(* POU STP, ST *)
PROGRAM STP
VAR
	LSL100A_MixerFloatSensor AT %I* : BOOL;
	LSH100A_MixerFloatSensor AT %I* : BOOL;
	LSH101A_EQFloatSensor AT %I* : BOOL;
	LSHH101A_EQFloatSensor AT %I* : BOOL;
	LSL101A_EQFloatSensor AT %I* : BOOL;
	LSH105A1_StreamLineFlow AT %I* : BOOL;
	LSHH105A2_StreamLineOverflow AT %I* : BOOL;
	LSL103A_SBRFloatSensor AT %I* : BOOL;
	LSHH103A_SBRFloatSensor AT %I* : BOOL;
	LSH103A_SBRFloatSensor AT %I* : BOOL;
	TMT01_FanStatus AT %I* : BOOL;
	DP01_DoorPanelStatus AT %I* : BOOL;
	LSD101A_EQFloatSensorDry AT %I* : BOOL;
	LSD103A_SBRFloatSensorDry AT %I* : BOOL;
	XV101A1_SolenoidValveSpray_OpenStat AT %I* : BOOL;
	XV101A2_SolenoidValveSpray_OpenStat AT %I* : BOOL;
	XV102A1_ContinuosValveWater_OpenStat AT %I* : BOOL;
	XV100A1_GritRemovalValve_OpenStat AT %I* : BOOL;
	XV100A2_GritRemovalValve_OpenStat AT %I* : BOOL;
	PS101A1_Penstock_OpenStat AT %I* : BOOL;
	PS101A2_Penstock_OpenStat AT %I* : BOOL;
	PS101A1_Penstock_CloseStat AT %I* : BOOL;
	PS101A2_Penstock_CloseStat AT %I* : BOOL;
	XV101A1_SolenoidValveSpray_CloseStat AT %I* : BOOL;
	XV101A2_SolenoidValveSpray_CloseStat AT %I* : BOOL;
	XV102A1_ContinuosValveWater_CloseStat AT %I* : BOOL;
	XV100A1_GritRemovalValve_CloseStat AT %I* : BOOL;
	XV100A2_GritRemovalValve_CloseStat AT %I* : BOOL;
	M101A1_EQMixer_OverloadStat AT %I* : BOOL;
	M101A1_EQMixer_IncompleteStat AT %I* : BOOL;
	M101A2_EQMixer_OverloadStat AT %I* : BOOL;
	M101A2_EQMixer_IncompleteStat AT %I* : BOOL;
	P101A1_EQPump_OverloadStat AT %I* : BOOL;
	P101A1_EQPump_IncompleteStat AT %I* : BOOL;
	P101A2_EQPump_OverloadStat AT %I* : BOOL;
	P101A2_EQPump_IncompleteStat AT %I* : BOOL;
	PS101A1_Penstock_TripStat AT %I* : BOOL;
	PS101A2_Penstock_TripStat AT %I* : BOOL;
	F101A1_FineScr_OverloadStat AT %I* : BOOL;
	F101A2_FineScr_OverloadStat AT %I* : BOOL;
	C102A_ScreeningConveyer_OverloadStat AT %I* : BOOL;
	C101A_ScreeningCompactor_OverloadStat AT %I* : BOOL;
	C103A_GritClassifier_OverloadStat AT %I* : BOOL;
	P102A1_SBRTransferPump_OverloadStat AT %I* : BOOL;
	P102A1_SBRTransferPump_IncompleteStat AT %I* : BOOL;
	P102A2_SBRTransferPump_OverloadStat AT %I* : BOOL;
	P102A2_SBRTransferPump_IncompleteStat AT %I* : BOOL;
	M101A1_EQMixer_LocalRemoteStat AT %I* : BOOL;
	M101A2_EQMixer_LocalRemoteStat AT %I* : BOOL;
	P101A1_EQPump_LocalRemoteStat AT %I* : BOOL;
	P101A2_EQPump_LocalRemoteStat AT %I* : BOOL;
	F101A1_FineScr_LocalRemoteStat AT %I* : BOOL;
	F101A2_FineScr_LocalRemoteStat AT %I* : BOOL;
	C102A_ScreenConveyer_LocalRemoteStat AT %I* : BOOL;
	C101A_ScreenCompactor_LocalRemoteStat AT %I* : BOOL;
	C103A_GritClasifier_LocalRemoteStat AT %I* : BOOL;
	P102A1_SBRTransferPump_LocalRemoteStat AT %I* : BOOL;
	P102A2_SBRTransferPump_LocalRemoteStat AT %I* : BOOL;
	PS101A1_Penstock_LocalRemoteStat AT %I* : BOOL;
	PS101A2_Penstock_LocalRemoteStat AT %I* : BOOL;
	M101A1_EQMixer_RunStat AT %I* : BOOL;
	M101A2_EQMixer_RunStat AT %I* : BOOL;
	P101A1_EQPump_RunStat AT %I* : BOOL;
	P101A2_EQPump_RunStat AT %I* : BOOL;
	F101A1_FineScr_RunStat AT %I* : BOOL;
	F101A2_FineScr_RunStat AT %I* : BOOL;
	C102A_ScreenConveyer_RunStat AT %I* : BOOL;
	C101A_ScreenCompactor_RunStat AT %I* : BOOL;
	C103A_GritClasifier_RunStat AT %I* : BOOL;
	P102A1_SBRTransferPump_RunStat AT %I* : BOOL;
	P102A2_SBRTransferPump_RunStat AT %I* : BOOL;
	M101A1_EQMixer_EStopStat AT %I* : BOOL;
	M101A2_EQMixer_EStopStat AT %I* : BOOL;
	P101A1_EQPump_EStopStat AT %I* : BOOL;
	P101A2_EQPump_EStopStat AT %I* : BOOL;
	F101A1_FineScr_EStopStat AT %I* : BOOL;
	F101A2_FineScr_EStopStat AT %I* : BOOL;
	C102A_ScreenConveyer_EStopStat AT %I* : BOOL;
	C101A_ScreenCompactor_EStopStat AT %I* : BOOL;
	C103A_GritClasifier_EStopStat AT %I* : BOOL;
	P102A1_SBRTransferPump_EStopStat AT %I* : BOOL;
	P102A2_SBRTransferPump_EStopStat AT %I* : BOOL;
	B101A1_AirBlower_OverloadStat AT %I* : BOOL;
	B101A1_AirBlower_IncompleteStat AT %I* : BOOL;
	B101A2_AirBlower_OverloadStat AT %I* : BOOL;
	B101A2_AirBlower_IncompleteStat AT %I* : BOOL;
	B101A1_AirBlower_LocalRemoteStat AT %I* : BOOL;
	B101A2_AirBlower_LocalRemoteStat AT %I* : BOOL;
	B101A1_AirBlower_OnOffStat AT %I* : BOOL;
	B101A2_AirBlower_OnOffStat AT %I* : BOOL;
	B101A1_AirBlower_EStopStat AT %I* : BOOL;
	B101A2_AirBlower_EStopStat AT %I* : BOOL;
	XV101A1_SolenoidValveSpray_OpenCmd AT %Q* : BOOL;
	XV101A2_SolenoidValveSpray_OpenCmd AT %Q* : BOOL;
	XV102A1_ContinuosValveWater_OpenCmd AT %Q* : BOOL;
	F101A1_FineScr_RunCmd AT %Q* : BOOL;
	F101A2_FineScr_RunCmd AT %Q* : BOOL;
	C102A_ScreenConveyer_RunCmd AT %Q* : BOOL;
	C101A_ScreenCompactor_RunCmd AT %Q* : BOOL;
	C103A_GritClasifier_RunCmd AT %Q* : BOOL;
	PS101A1_Penstock_OpenCmd AT %Q* : BOOL;
	PS101A1_Penstock_CloseCmd AT %Q* : BOOL;
	PS101A2_Penstock_OpenCmd AT %Q* : BOOL;
	PS101A2_Penstock_CloseCmd AT %Q* : BOOL;
	XV100A1_GritRemovalValve_OpenCmd AT %Q* : BOOL;
	XV100A2_GritRemovalValve_OpenCmd AT %Q* : BOOL;
	P101A1_EQPump_RunCmd AT %Q* : BOOL;
	P101A2_EQPump_RunCmd AT %Q* : BOOL;
	M101A1_EQMixer_RunCmd AT %Q* : BOOL;
	M101A2_EQMixer_RunCmd AT %Q* : BOOL;
	B101A1_AirBlower_RunCmd AT %Q* : BOOL;
	B101A2_AirBlower_RunCmd AT %Q* : BOOL;
	P102A1_SBRTransferPump_RunCmd AT %Q* : BOOL;
	P102A2_SBRTransferPump_RunCmd AT %Q* : BOOL;
	AUX101A_EQFloatSensor_AlarmS1 AT %Q* : BOOL;
	AUX104A_SBRFloatSensor_AlarmS1 AT %Q* : BOOL;
	AUX105A_StreamSensorOverflow_AlarmS1 AT %Q* : BOOL;
	AUX101_CommonAlarm AT %Q* : BOOL;
	AUX102_PLCRunStat AT %Q* : BOOL;
	LSL100B_MixerFloatSensor AT %I* : BOOL;
	LSH100B_MixerFloatSensor AT %I* : BOOL;
	LSH101B_EQFloatSensor AT %I* : BOOL;
	LSHH101B_EQFloatSensor AT %I* : BOOL;
	LSL101B_EQFloatSensor AT %I* : BOOL;
	LSH105B1_StreamLineFlow AT %I* : BOOL;
	LSHH105B2_StreamLineOverflow AT %I* : BOOL;
	LSH103B_SBRFloatSensor AT %I* : BOOL;
	LSHH103B_SBRFloatSensor AT %I* : BOOL;
	LSL103B_SBRFloatSensor AT %I* : BOOL;
	LSD101B_EQFloatSensorDry AT %I* : BOOL;
	LSD103B_SBRFloatSensorDry AT %I* : BOOL;
	XV101B1_SolenoidValveSpray_OpenStat AT %I* : BOOL;
	XV101B2_SolenoidValveSpray_OpenStat AT %I* : BOOL;
	XV102B1_ContinuosValveWater_OpenStat AT %I* : BOOL;
	XV100B1_GritRemovalValve_OpenStat AT %I* : BOOL;
	XV100B2_GritRemovalValve_OpenStat AT %I* : BOOL;
	PS101B1_Penstock_OpenStat AT %I* : BOOL;
	PS101B2_Penstock_OpenStat AT %I* : BOOL;
	PS101B1_Penstock_CloseStat AT %I* : BOOL;
	PS101B2_Penstock_CloseStat AT %I* : BOOL;
	XV101B1_SolenoidValveSpray_CloseStat AT %I* : BOOL;
	XV101B2_SolenoidValveSpray_CloseStat AT %I* : BOOL;
	XV102B1_ContinuosValveWater_CloseStat AT %I* : BOOL;
	XV100B1_GritRemovalValve_CloseStat AT %I* : BOOL;
	XV100B2_GritRemovalValve_CloseStat AT %I* : BOOL;
	M101B1_EQMixer_OverloadStat AT %I* : BOOL;
	M101B1_EQMixer_IncompleteStat AT %I* : BOOL;
	M101B2_EQMixer_OverloadStat AT %I* : BOOL;
	M101B2_EQMixer_IncompleteStat AT %I* : BOOL;
	P101B1_EQPump_OverloadStat AT %I* : BOOL;
	P101B1_EQPump_IncompleteStat AT %I* : BOOL;
	P101B2_EQPump_OverloadStat AT %I* : BOOL;
	P101B2_EQPump_IncompleteStat AT %I* : BOOL;
	PS101B1_Penstock_TripStat AT %I* : BOOL;
	PSB101B2_Penstock_TripStat AT %I* : BOOL;
	F101B1_FineScr_OverloadStat AT %I* : BOOL;
	F101B2_FineScr_OverloadStat AT %I* : BOOL;
	C102B_ScreeningConveyer_OverloadStat AT %I* : BOOL;
	C101B_ScreeningCompactor_OverloadStat AT %I* : BOOL;
	C103B_GritClassifier_OverloadStat AT %I* : BOOL;
	P102B1_SBRTransferPump_OverloadStat AT %I* : BOOL;
	P102B1_SBRTransferPump_IncompleteStat AT %I* : BOOL;
	P102B2_SBRTransferPump_OverloadStat AT %I* : BOOL;
	P102B2_SBRTransferPump_IncompleteStat AT %I* : BOOL;
	M101B1_EQMixer_LocalRemoteStat AT %I* : BOOL;
	M101B2_EQMixer_LocalRemoteStat AT %I* : BOOL;
	P101B1_EQPump_LocalRemoteStat AT %I* : BOOL;
	P101B2_EQPump_LocalRemoteStat AT %I* : BOOL;
	F101B1_FineScr_LocalRemoteStat AT %I* : BOOL;
	F101B2_FineScr_LocalRemoteStat AT %I* : BOOL;
	C102B_ScreenConveyer_LocalRemoteStat AT %I* : BOOL;
	C101B_ScreenCompactor_LocalRemoteStat AT %I* : BOOL;
	C103BB_GritClasifiier_LocalRemoteStat AT %I* : BOOL;
	P102B1_SBRTransferPump_LocalRemoteStat AT %I* : BOOL;
	P102B2_SBRTransferPump_LocalRemoteStat AT %I* : BOOL;
	PS101B1_Penstock_LocalRemoteStat AT %I* : BOOL;
	PS101B2_Penstock_LocalRemoteStat AT %I* : BOOL;
	M101B1_EQMixer_RunStat AT %I* : BOOL;
	M101B2_EQMixer_RunStat AT %I* : BOOL;
	P101B1_EQPump_RunStat AT %I* : BOOL;
	P101B2_EQPump_RunStat AT %I* : BOOL;
	F101B1_FineScr_RunStat AT %I* : BOOL;
	F101B2_FineScr_RunStat AT %I* : BOOL;
	C102B_ScreenConveyer_RunStat AT %I* : BOOL;
	C101B_ScreenCompactor_RunStat AT %I* : BOOL;
	C103B_GritClasifier_RunStat AT %I* : BOOL;
	P102B1_SBRTransferPump_RunStat AT %I* : BOOL;
	P102B2_SBRTransferPump_RunStat AT %I* : BOOL;
	M101B1_EQMixer_EStopStat AT %I* : BOOL;
	M101B2_EQMixer_EStopStat AT %I* : BOOL;
	P101B1_EQPump_EStopStat AT %I* : BOOL;
	P101B2_EQPump_EStopStat AT %I* : BOOL;
	F101B1_FineScr_EStopStat AT %I* : BOOL;
	F101B2_FineScr_EStopStat AT %I* : BOOL;
	C102B_ScreenConveyer_EStopStat AT %I* : BOOL;
	C101B_ScreenCompactor_EStopStat AT %I* : BOOL;
	C103B_GritClasifier_EStopStat AT %I* : BOOL;
	P102B1_SBRTransferPump_EStopStat AT %I* : BOOL;
	P102B2_SBRTransferPump_EStopStat AT %I* : BOOL;
	VE801A_SuctionFan_OnOffStat AT %I* : BOOL;
	P802A_CirculationPump_OnOffStat AT %I* : BOOL;
	P803A_CirculationPump_OnOffStat AT %I* : BOOL;
	P804A_CirculationPump_OnOffStat AT %I* : BOOL;
	P805A1_H2S04Pump_OnOffStat AT %I* : BOOL;
	P805A2_H2S04Pump_OnOffStat AT %I* : BOOL;
	P806A1_NAOHPump_OnOffStat AT %I* : BOOL;
	P806A2_NAOHPump_OnOffStat AT %I* : BOOL;
	P807A1_NAOCLPump_OnOffStat AT %I* : BOOL;
	P807A2_NAOCLPump_OnOffStat AT %I* : BOOL;
	VE801A_SuctionFan_OverloadStat AT %I* : BOOL;
	P802A_CirculationPump_OverloadStat AT %I* : BOOL;
	P803A_CirculationPump_OverloadStat AT %I* : BOOL;
	P804A_CirculationPump_OverloadStat AT %I* : BOOL;
	P805A1_H2S04Pump_OverloadStat AT %I* : BOOL;
	P805A2_H2S04Pump_OverloadStat AT %I* : BOOL;
	P806A1_NAOHPump_OverloadStat AT %I* : BOOL;
	P806A2_NAOHPump_OverloadStat AT %I* : BOOL;
	P807A1_NAOCLPump_OverloadStat AT %I* : BOOL;
	P807A2_NAOCLPump_OverloadStat AT %I* : BOOL;
	VE801A_SuctionFan_EStopStat AT %I* : BOOL;
	P802A_CirculationPump_EStopStat AT %I* : BOOL;
	P803A_CirculationPump_EStopStat AT %I* : BOOL;
	P804A_CirculationPump_EStopStat AT %I* : BOOL;
	P805A1_H2S04Pump_EStopStat AT %I* : BOOL;
	P805A2_H2S04Pump_EStopStat AT %I* : BOOL;
	P806A1_NAOHPump_EStopStat AT %I* : BOOL;
	P806A2_NAOHPump_EStopStat AT %I* : BOOL;
	P807A1_NAOCLPump_EStopStat AT %I* : BOOL;
	P807A2_NAOCLPump_EStopStat AT %I* : BOOL;
	XV101B1_SolenoidValveSpray_OpenCmd AT %Q* : BOOL;
	XV101B2_SolenoidValveSpray_OpenCmd AT %Q* : BOOL;
	XV102B1_ContinuosValveWater_OpenCmd AT %Q* : BOOL;
	F101B1_FineScr_RunCmd AT %Q* : BOOL;
	F101B2_FineScr_RunCmd AT %Q* : BOOL;
	C102B_ScreenConveyer_RunCmd AT %Q* : BOOL;
	C101B_ScreenCompactor_RunCmd AT %Q* : BOOL;
	C103B_GritClasifier_RunCmd AT %Q* : BOOL;
	PS101B1_Penstock_OpenCmd AT %Q* : BOOL;
	PS101B1_Penstock_CloseCmd AT %Q* : BOOL;
	PS101B2_Penstock_OpenCmd AT %Q* : BOOL;
	PS101B2_Penstock_CloseCmd AT %Q* : BOOL;
	XV100B1_GritRemovalValve_OpenCmd AT %Q* : BOOL;
	XV100B2_GritRemovalValve_OpenCmd AT %Q* : BOOL;
	P101B1_EQPump_RunCmd AT %Q* : BOOL;
	P101B2_EQPump_RunCmd AT %Q* : BOOL;
	M101B1_EQMixer_RunCmd AT %Q* : BOOL;
	M101B2_EQMixer_RunCmd AT %Q* : BOOL;
	P102B1_SBRTransferPump_RunCmd AT %Q* : BOOL;
	P102B2_SBRTransferPump_RunCmd AT %Q* : BOOL;
	AUX101B_EQFloatSensor_AlarmS2 AT %Q* : BOOL;
	AUX104B_SBRFloatSensor_AlarmS2 AT %Q* : BOOL;
	AUX105B_StreamSensorOverflow_AlarmS2 AT %Q* : BOOL;
	TMT02_FanStatus AT %I* : BOOL;
	DP02_DoorPanelStatus AT %I* : BOOL;
	XV261A_DecanterR1_OverloadStat AT %I* : BOOL;
	XV262A_DecanterR2_OverloadStat AT %I* : BOOL;
	XV263A_DecanterR3_OverloadStat AT %I* : BOOL;
	XV264A_DecanterR4_OverloadStat AT %I* : BOOL;
	M200A1A_MixerR1_RunStat AT %I* : BOOL;
	M200A1B_MixerR1_RunStat AT %I* : BOOL;
	M200A1C_MixerR1_RunStat AT %I* : BOOL;
	M200A2A_MixerR2_RunStat AT %I* : BOOL;
	M200A2B_MixerR2_RunStat AT %I* : BOOL;
	M200A2C_MixerR2_RunStat AT %I* : BOOL;
	M200A3A_MixerR3_RunStat AT %I* : BOOL;
	M200A3B_MixerR3_RunStat AT %I* : BOOL;
	M200A3C_MixerR3_RunStat AT %I* : BOOL;
	M200A4A_MixerR4_RunStat AT %I* : BOOL;
	M200A4B_MixerR4_RunStat AT %I* : BOOL;
	M200A4C_MixerR4_RunStat AT %I* : BOOL;
	B201A1_AirBlowerS1_RunStat AT %I* : BOOL;
	B201A2_AirBlowerS1_RunStat AT %I* : BOOL;
	B201A3_AirBlowerS1_RunStat AT %I* : BOOL;
	M200A1A_MixerR1_LocalRemoteStat AT %I* : BOOL;
	M200A1B_MixerR1_LocalRemoteStat AT %I* : BOOL;
	M200A1C_MixerR1_LocalRemoteStat AT %I* : BOOL;
	M200A2A_MixerR2_LocalRemoteStat AT %I* : BOOL;
	M200A2B_MixerR2_LocalRemoteStat AT %I* : BOOL;
	M200A2C_MixerR2_LocalRemoteStat AT %I* : BOOL;
	M200A3A_MixerR3_LocalRemoteStat AT %I* : BOOL;
	M200A3B_MixerR3_LocalRemoteStat AT %I* : BOOL;
	M200A3C_MixerR3_LocalRemoteStat AT %I* : BOOL;
	M200A4A_MixerR4_LocalRemoteStat AT %I* : BOOL;
	M200A4B_MixerR4_LocalRemoteStat AT %I* : BOOL;
	M200A4C_MixerR4_LocalRemoteStat AT %I* : BOOL;
	B201A1_AirBlowerS1_LocalRemoteStat AT %I* : BOOL;
	B201A2_AirBlowerS1_LocalRemoteStat AT %I* : BOOL;
	B201A3_AirBlowerS1_LocalRemoteStat AT %I* : BOOL;
	XV261A_DecanterR1_LocalRemoteStat AT %I* : BOOL;
	XV262A_DecanterR2_LocalRemoteStat AT %I* : BOOL;
	XV263A_DecanterR3_LocalRemoteStat AT %I* : BOOL;
	XV264A_DecanterR4_LocalRemoteStat AT %I* : BOOL;
	P201A1_DesludgePumpS1_LocalRemoteStat AT %I* : BOOL;
	P201A2_DesludgePumpS1_LocalRemoteStat AT %I* : BOOL;
	P201A1_DesludgePumpS1_RunStat AT %I* : BOOL;
	P201A2_DesludgePumpS1_RunStat AT %I* : BOOL;
	M200A1A_MixerR1_OverloadStat AT %I* : BOOL;
	M200A1A_MixerR1_IncompleteStat AT %I* : BOOL;
	M200A1B_MixerR1_OverloadStat AT %I* : BOOL;
	M200A1B_MixerR1_IncompleteStat AT %I* : BOOL;
	M200A1C_MixerR1_OverloadStat AT %I* : BOOL;
	M200A1C_MixerR1_IncompleteStat AT %I* : BOOL;
	M200A2A_MixerR2_OverloadStat AT %I* : BOOL;
	M200A2A_MixerR2_IncompleteStat AT %I* : BOOL;
	M200A2B_MixerR2_OverloadStat AT %I* : BOOL;
	M200A2B_MixerR2_IncompleteStat AT %I* : BOOL;
	M200A2C_MixerR2_OverloadStat AT %I* : BOOL;
	M200A2C_MixerR2_IncompleteStat AT %I* : BOOL;
	M200A3A_MixerR3_OverloadStat AT %I* : BOOL;
	M200A3A_MixerR3_IncompleteStat AT %I* : BOOL;
	M200A3B_MixerR3_OverloadStat AT %I* : BOOL;
	M200A3B_MixerR3_IncompleteStat AT %I* : BOOL;
	M200A3C_MixerR3_OverloadStat AT %I* : BOOL;
	M200A3C_MixerR3_IncompleteStat AT %I* : BOOL;
	M200A4A_MixerR4_OverloadStat AT %I* : BOOL;
	M200A4A_MixerR4_IncompleteStat AT %I* : BOOL;
	M200A4B_MixerR4_OverloadStat AT %I* : BOOL;
	M200A4B_MixerR4_IncompleteStat AT %I* : BOOL;
	M200A4C_MixerR4_OverloadStat AT %I* : BOOL;
	M200A4C_MixerR4_IncompleteStat AT %I* : BOOL;
	B201A1_AirBlowerS1_OverloadStat AT %I* : BOOL;
	B201A1_AirBlowerS1_IncompleteStat AT %I* : BOOL;
	B201A2_AirBlowerS1_OverloadStat AT %I* : BOOL;
	B201A2_AirBlowerS1_IncompleteStat AT %I* : BOOL;
	B201A3_AirBlowerS1_OverloadStat AT %I* : BOOL;
	B201A3_AirBlowerS1_IncompleteStat AT %I* : BOOL;
	P201A1_DesludgePumpS1_OverloadStatus AT %I* : BOOL;
	P201A2_DesludgePumpS1_OverloadStatus AT %I* : BOOL;
	M200A1A_MixerR1_EStopStat AT %I* : BOOL;
	M200A1B_MixerR1_EStopStat AT %I* : BOOL;
	M200A1C_MixerR1_EStopStat AT %I* : BOOL;
	M200A2A_MixerR2_EStopStat AT %I* : BOOL;
	M200A2B_MixerR2_EStopStat AT %I* : BOOL;
	M200A2C_MixerR2_EStopStat AT %I* : BOOL;
	M200A3A_MixerR3_EStopStat AT %I* : BOOL;
	M200A3B_MixerR3_EStopStat AT %I* : BOOL;
	M200A3C_MixerR3_EStopStat AT %I* : BOOL;
	M200A4A_MixerR3_EStopStat AT %I* : BOOL;
	M200A4B_MixerR3_EStopStat AT %I* : BOOL;
	M200A4C_MixerR3_EStopStat AT %I* : BOOL;
	B201A1_AirBlowerS1_EStopStat AT %I* : BOOL;
	B201A2_AirBlowerS1_EStopStat AT %I* : BOOL;
	B201A3_AirBlowerS1_EStopStat AT %I* : BOOL;
	XV261A_DecanterR1_EStopStat AT %I* : BOOL;
	XV262A_DecanterR2_EStopStat AT %I* : BOOL;
	XV263A_DecanterR3_EStopStat AT %I* : BOOL;
	XV264A_DecanterR4_EStopStat AT %I* : BOOL;
	P201A1_DesludgePumpS1_EStopStat AT %I* : BOOL;
	P201A2_DesludgePumpS1_EStopStat AT %I* : BOOL;
	XV261A_DecanterR1_FwdStat AT %I* : BOOL;
	XV262A_DecanterR2_FwdStat AT %I* : BOOL;
	XV263A_DecanterR3_FwdStat AT %I* : BOOL;
	XV264A_DecanterR4_FwdStat AT %I* : BOOL;
	XV261A_DecanterR1_RvsStat AT %I* : BOOL;
	XV262A_DecanterR2_RvsStat AT %I* : BOOL;
	XV263A_DecanterR3_RvsStat AT %I* : BOOL;
	XV264A_DecanterR4_RvsStat AT %I* : BOOL;
	FT100A_FlowTotalizerS1 AT %IW0 : REAL;
	FT100A_FlowTotalizerS1_ScaledValue:INT;
	M200A1A_MixerR1_RunCmd AT %Q* : BOOL;
	M200A1B_MixerR1_RunCmd AT %Q* : BOOL;
	M200A1C_MixerR1_RunCmd AT %Q* : BOOL;
	M200A2A_MixerR2_RunCmd AT %Q* : BOOL;
	M200A2B_MixerR2_RunCmd AT %Q* : BOOL;
	M200A2C_MixerR2_RunCmd AT %Q* : BOOL;
	M200A3A_MixerR3_RunCmd AT %Q* : BOOL;
	M200A3B_MixerR3_RunCmd AT %Q* : BOOL;
	M200A3C_MixerR3_RunCmd AT %Q* : BOOL;
	M200A4A_MixerR4_RunCmd AT %Q* : BOOL;
	M200A4B_MixerR4_RunCmd AT %Q* : BOOL;
	M200A4C_MixerR4_RunCmd AT %Q* : BOOL;
	XV261A_DecanterR1_FwdCmd AT %Q* : BOOL;
	XV262A_DecanterR2_FwdCmd AT %Q* : BOOL;
	XV263A_DecanterR3_FwdCmd AT %Q* : BOOL;
	XV264A_DecanterR4_FwdCmd AT %Q* : BOOL;
	XV261A_DecanterR1_RvsCmd AT %Q* : BOOL;
	XV262A_DecanterR2_RvsCmd AT %Q* : BOOL;
	XV263A_DecanterR3_RvsCmd AT %Q* : BOOL;
	XV264A_DecanterR4_RvsCmd AT %Q* : BOOL;
	B201A1_AirBlowerS1_RunCmd AT %Q* : BOOL;
	B201A2_AirBlowerS1_RunCmd AT %Q* : BOOL;
	B201A3_AirBlowerS1_RunCmd AT %Q* : BOOL;
	P201A1_DesludgePump_RunCmd AT %Q* : BOOL;
	P201A2_DesludgePump_RunCmd AT %Q* : BOOL;
	AUXA1_ReactorS1R1_OpsStat AT %Q* : BOOL;
	AUXA2_ReactorS1R2_OpsStat AT %Q* : BOOL;
	AUXA3_ReactorS1R3_OpsStat AT %Q* : BOOL;
	AUXA4_ReactorS1R4_OpsStat AT %Q* : BOOL;
	AUXB1_ReactorS2R1_OpsStat AT %Q* : BOOL;
	AUXB2_ReactorS2R2_OpsStat AT %Q* : BOOL;
	AUXB3_ReactorS2R3_OpsStat AT %Q* : BOOL;
	AUXB4_ReactorS2R4_OpsStat AT %Q* : BOOL;
	AUXA5_BlowerS1R1 AT %Q* : BOOL;
	AUXA6_BlowerS1R2 AT %Q* : BOOL;
	AUXA7_BlowerS1R3 AT %Q* : BOOL;
	AUXB5_BlowerS2R1 AT %Q* : BOOL;
	AUXB6_BlowerS2R2 AT %Q* : BOOL;
	AUXB7_BlowerS2R3 AT %Q* : BOOL;
	AUX201_CommonAlarm AT %Q* : BOOL;
	AUX202_PLCRunStat AT %Q* : BOOL;
	TMT03_FanStatus AT %I* : BOOL;
	DP03_DoorPanelStatus AT %I* : BOOL;
	XV261B_DecanterR1_OverloadStat AT %I* : BOOL;
	XV262B_DecanterR2_OverloadStat AT %I* : BOOL;
	XV263B_DecanterR3_OverloadStat AT %I* : BOOL;
	XV264B_DecanterR4_OverloadStat AT %I* : BOOL;
	M200B1A_MixerR1_RunStat AT %I* : BOOL;
	M200B1B_MixerR1_RunStat AT %I* : BOOL;
	M200B1C_MixerR1_RunStat AT %I* : BOOL;
	M200B2A_MixerR2_RunStat AT %I* : BOOL;
	M200B2B_MixerR2_RunStat AT %I* : BOOL;
	M200B2C_MixerR2_RunStat AT %I* : BOOL;
	M200B3A_MixerR3_RunStat AT %I* : BOOL;
	M200B3B_MixerR3_RunStat AT %I* : BOOL;
	M200B3C_MixerR3_RunStat AT %I* : BOOL;
	M200B4A_MixerR4_RunStat AT %I* : BOOL;
	M200B4B_MixerR4_RunStat AT %I* : BOOL;
	M200B4C_MixerR4_RunStat AT %I* : BOOL;
	B201B1_AirBlowerS2_RunStat AT %I* : BOOL;
	B201B2_AirBlowerS2_RunStat AT %I* : BOOL;
	B201B3_AirBlowerS2_RunStat AT %I* : BOOL;
	M200B1A_MixerR1_LocalRemoteStat AT %I* : BOOL;
	M200B1B_MixerR1_LocalRemoteStat AT %I* : BOOL;
	M200B1C_MixerR1_LocalRemoteStat AT %I* : BOOL;
	M200B2A_MixerR2_LocalRemoteStat AT %I* : BOOL;
	M200B2B_MixerR2_LocalRemoteStat AT %I* : BOOL;
	M200B2C_MixerR2_LocalRemoteStat AT %I* : BOOL;
	M200B3A_MixerR3_LocalRemoteStat AT %I* : BOOL;
	M200B3B_MixerR3_LocalRemoteStat AT %I* : BOOL;
	M200B3C_MixerR3_LocalRemoteStat AT %I* : BOOL;
	M200B4A_MixerR4_LocalRemoteStat AT %I* : BOOL;
	M200B4B_MixerR4_LocalRemoteStat AT %I* : BOOL;
	M200B4C_MixerR4_LocalRemoteStat AT %I* : BOOL;
	B201B1_AirBlowerS2_LocalRemoteStat AT %I* : BOOL;
	B201B2_AirBlowerS2_LocalRemoteStat AT %I* : BOOL;
	B201B3_AirBlowerS2_LocalRemoteStat AT %I* : BOOL;
	XV261B_DecanterR1_LocalRemoteStat AT %I* : BOOL;
	XV262B_DecanterR2_LocalRemoteStat AT %I* : BOOL;
	XV263B_DecanterR3_LocalRemoteStat AT %I* : BOOL;
	XV264B_DecanterR4_LocalRemoteStat AT %I* : BOOL;
	P201B1_DesludgePumpS2_LocalRemoteStat AT %I* : BOOL;
	P201B2_DesludgePumpS2_LocalRemoteStat AT %I* : BOOL;
	P201B1_DesludgePumpS2_RunStat AT %I* : BOOL;
	P201B2_DesludgePumpS2_RunStat AT %I* : BOOL;
	M200B1A_MixerR1_OverloadStat AT %I* : BOOL;
	M200B1A_MixerR1_IncompleteStat AT %I* : BOOL;
	M200B1B_MixerR1_OverloadStat AT %I* : BOOL;
	M200B1B_MixerR1_IncompleteStat AT %I* : BOOL;
	M200B1C_MixerR1_OverloadStat AT %I* : BOOL;
	M200B1C_MixerR1_IncompleteStat AT %I* : BOOL;
	M200B2A_MixerR2_OverloadStat AT %I* : BOOL;
	M200B2A_MixerR2_IncompleteStat AT %I* : BOOL;
	M200B2B_MixerR2_OverloadStat AT %I* : BOOL;
	M200B2B_MixerR2_IncompleteStat AT %I* : BOOL;
	M200B2C_MixerR2_OverloadStat AT %I* : BOOL;
	M200B2C_MixerR2_IncompleteStat AT %I* : BOOL;
	M200B3A_MixerR3_OverloadStat AT %I* : BOOL;
	M200B3A_MixerR2_IncompleteStat AT %I* : BOOL;
	M200B3B_MixerR3_OverloadStat AT %I* : BOOL;
	M200B3B_MixerR3_IncompleteStat AT %I* : BOOL;
	M200B3C_MixerR3_OverloadStat AT %I* : BOOL;
	M200B3C_MixerR3_IncompleteStat AT %I* : BOOL;
	M200B4A_MixerR4_OverloadStat AT %I* : BOOL;
	M200B4A_MixerR4_IncompleteStat AT %I* : BOOL;
	M200B4B_MixerR4_OverloadStat AT %I* : BOOL;
	M200B4B_MixerR4_IncompleteStat AT %I* : BOOL;
	M200B4C_MixerR4_OverloadStat AT %I* : BOOL;
	M200B4C_MixerR4_IncompleteStat AT %I* : BOOL;
	B201B1_AirBlowerS2_OverloadStat AT %I* : BOOL;
	B201B1_AirBlowerS2_IncompleteStat AT %I* : BOOL;
	B201B2_AirBlowerS2_OverloadStat AT %I* : BOOL;
	B201B2_AirBlowerS2_IncompleteStat AT %I* : BOOL;
	B201B3_AirBlowerS2_OverloadStat AT %I* : BOOL;
	B201B3_AirBlowerS2_IncompleteStat AT %I* : BOOL;
	P201B1_DesludgePumpS2_OverloadStat AT %I* : BOOL;
	P201B2_DesludgePumpS2_OverloadStat AT %I* : BOOL;
	M200B1A_MixerR1_EStopStat AT %I* : BOOL;
	M200B1B_MixerR1_EStopStat AT %I* : BOOL;
	M200B1C_MixerR1_EStopStat AT %I* : BOOL;
	M200B2A_MixerR2_EStopStat AT %I* : BOOL;
	M200B2B_MixerR2_EStopStat AT %I* : BOOL;
	M200B2C_MixerR2_EStopStat AT %I* : BOOL;
	M200B3A_MixerR3_EStopStat AT %I* : BOOL;
	M200B3B_MixerR3_EStopStat AT %I* : BOOL;
	M200B3C_MixerR3_EStopStat AT %I* : BOOL;
	M200B4A_MixerR4_EStopStat AT %I* : BOOL;
	M200B4B_MixerR4_EStopStat AT %I* : BOOL;
	M200B4C_MixerR4_EStopStat AT %I* : BOOL;
	B201B1_AirBlowerS2_EStopStat AT %I* : BOOL;
	B201B2_AirBlowerS2_EStopStat AT %I* : BOOL;
	B201B3_AirBlowerS2_EStopStat AT %I* : BOOL;
	XV261B_DecanterR1_EStopStat AT %I* : BOOL;
	XV262B_DecanterR2_EStopStat AT %I* : BOOL;
	XV263B_DecanterR3_EStopStat AT %I* : BOOL;
	XV264B_DecanterR4_EStopStat AT %I* : BOOL;
	P201B1_DesludgePumpS2_EStopStat AT %I* : BOOL;
	P201B2_DesludgePumpS2_EStopStat AT %I* : BOOL;
	XV261B_DecanterR1_FwdStat AT %I* : BOOL;
	XV262B_DecanterR2_FwdStat AT %I* : BOOL;
	XV263B_DecanterR3_FwdStat AT %I* : BOOL;
	XV264B_DecanterR4_FwdStat AT %I* : BOOL;
	XV261B_DecanterR1_RvsStat AT %I* : BOOL;
	XV262B_DecanterR2_RvsStat AT %I* : BOOL;
	XV263B_DecanterR3_RvsStat AT %I* : BOOL;
	XV264B_DecanterR4_RvsStat AT %I* : BOOL;
	FT100B_FlowTotalizerS2 AT %IW0 : REAL;
	FT100B_FlowTotalizerS2_ScaledValue:INT;
	M200B1A_MixerR1_RunCmd AT %Q* : BOOL;
	M200B1B_MixerR1_RunCmd AT %Q* : BOOL;
	M200B1C_MixerR1_RunCmd AT %Q* : BOOL;
	M200B2A_MixerR2_RunCmd AT %Q* : BOOL;
	M200B2B_MixerR2_RunCmd AT %Q* : BOOL;
	M200B2C_MixerR2_RunCmd AT %Q* : BOOL;
	M200B3A_MixerR3_RunCmd AT %Q* : BOOL;
	M200B3B_MixerR3_RunCmd AT %Q* : BOOL;
	M200B3C_MixerR3_RunCmd AT %Q* : BOOL;
	M200B4A_MixerR4_RunCmd AT %Q* : BOOL;
	M200B4B_MixerR4_RunCmd AT %Q* : BOOL;
	M200B4C_MixerR4_RunCmd AT %Q* : BOOL;
	XV261B_DecanterR1_FwdCmd AT %Q* : BOOL;
	XV262B_DecanterR2_FwdCmd AT %Q* : BOOL;
	XV263B_DecanterR3_FwdCmd AT %Q* : BOOL;
	XV264B_DecanterR4_FwdCmd AT %Q* : BOOL;
	XV261B_DecanterR1_RvsCmd AT %Q* : BOOL;
	XV262B_DecanterR2_RvsCmd AT %Q* : BOOL;
	XV263B_DecanterR3_RvsCmd AT %Q* : BOOL;
	XV264B_DecanterR4_RvsCmd AT %Q* : BOOL;
	B201B1_AirBlowerS2_RunCmd AT %Q* : BOOL;
	B201B2_AirBlowerS2_RunCmd AT %Q* : BOOL;
	B201B3_AirBlowerS2_RunCmd AT %Q* : BOOL;
	P201B1_DesludgePumpS2_RunCmd AT %Q* : BOOL;
	P201B2_DesludgePumpS2_RunCmd AT %Q* : BOOL;
	LSH201A1_LevelSensorR1 AT %I* : BOOL;
	LSH201A2_LevelSensorR2 AT %I* : BOOL;
	LSH201A3_LevelSensorR3 AT %I* : BOOL;
	LSH201A4_LevelSensorR4 AT %I* : BOOL;
	OPR1A_ReactorStatus AT %I* : BOOL;
	OPR2A_ReactorStatus AT %I* : BOOL;
	OPR3A_ReactorStatus AT %I* : BOOL;
	OPR4A_ReactorStatus AT %I* : BOOL;
	DP04_DoorPanelStatus AT %I* : BOOL;
	TMT04_FanStatus AT %I* : BOOL;
	HR201A1_DecantHighLevelR1 AT %I* : BOOL;
	LR201A1_DecantLowLevelR1 AT %I* : BOOL;
	HR201A2_DecantHighLevelR2 AT %I* : BOOL;
	LR201A2_DecantLowLevelR2 AT %I* : BOOL;
	HR201A3_DecantHighLevelR3 AT %I* : BOOL;
	LR201A3_DecantLowLevelR3 AT %I* : BOOL;
	HR201A4_DecantHighLevelR4 AT %I* : BOOL;
	LR201A4_DecantLowLevelR4 AT %I* : BOOL;
	XV205A_SBRValveR1_OpenStat AT %I* : BOOL;
	XV206A_SBRValveR2_OpenStat AT %I* : BOOL;
	XV207A_SBRValveR3_OpenStat AT %I* : BOOL;
	XV208A_SBRValveR4_OpenStat AT %I* : BOOL;
	XV201A_AirBlowerValveR1_OpenStat AT %I* : BOOL;
	XV202A_AirBlowerValveR2_OpenStat AT %I* : BOOL;
	XV203A_AirBlowerValveR3_OpenStat AT %I* : BOOL;
	XV204A_AirBlowerValveR4_OpenStat AT %I* : BOOL;
	XV221A_LimeValveR1_OpenStat AT %I* : BOOL;
	XV222A_LimeValveR2_OpenStat AT %I* : BOOL;
	XV223A_LimeValveR3_OpenStat AT %I* : BOOL;
	XV224A_LimeValveR4_OpenStat AT %I* : BOOL;
	XV211A_AlumValveR1_OpenStat AT %I* : BOOL;
	XV212A_AlumValveR2_OpenStat AT %I* : BOOL;
	XV213A_AlumValveR3_OpenStat AT %I* : BOOL;
	XV214A_AlumValveR4_OpenStat AT %I* : BOOL;
	XV205A_SBRValveR1_CloseStat AT %I* : BOOL;
	XV206A_SBRValveR2_CloseStat AT %I* : BOOL;
	XV207A_SBRValveR3_CloseStat AT %I* : BOOL;
	XV208A_SBRValveR4_CloseStat AT %I* : BOOL;
	XV201A_AirBlowerValveR1_CloseStat AT %I* : BOOL;
	XV202A_AirBlowerValveR2_CloseStat AT %I* : BOOL;
	XV203A_AirBlowerValveR3_CloseStat AT %I* : BOOL;
	XV204A_AirBlowerValveR4_CloseStat AT %I* : BOOL;
	XV221A_LimeValveR1_CloseStat AT %I* : BOOL;
	XV222A_LimeValveR2_CloseStat AT %I* : BOOL;
	XV223A_LimeValveR3_CloseStat AT %I* : BOOL;
	XV224A_LimeValveR4_CloseStat AT %I* : BOOL;
	XV211A_AlumValveR1_CloseStat AT %I* : BOOL;
	XV212A_AlumValveR2_CloseStat AT %I* : BOOL;
	XV213A_AlumValveR3_CloseStat AT %I* : BOOL;
	XV214A_AlumValveR4_CloseStat AT %I* : BOOL;
	XV241A_SludgeValveR1_CloseStat AT %I* : BOOL;
	XV242A_SludgeValveR2_CloseStat AT %I* : BOOL;
	XV243A_SludgeValveR3_CloseStat AT %I* : BOOL;
	XV244A_SludgeValveR4_CloseStat AT %I* : BOOL;
	XV241A_SludgeValveR1_OpenStat AT %I* : BOOL;
	XV242A_SludgeValveR2_OpenStat AT %I* : BOOL;
	XV243A_SludgeValveR3_OpenStat AT %I* : BOOL;
	XV244A_SludgeValveR4_OpenStat AT %I* : BOOL;
	D0201A4_DOProfilesR4 AT %IW0 : REAL;
	D0201A4_DOProfilesR4_ScaledValue:INT;
	DO201A1_DOProfilesR1 AT %IW0 : REAL;
	DO201A1_DOProfilesR1_ScaledValue:INT;
	DO201A2_DOProfilesR2 AT %IW0 : REAL;
	DO201A2_DOProfilesR2_ScaledValue:INT;
	DO201A3_DOProfilesR3 AT %IW0 : REAL;
	DO201A3_DOProfilesR3_ScaledValue:INT;
	PHT201A1_pHlevelR1 AT %IW0 : REAL;
	PHT201A1_pHlevelR1_ScaledValue:INT;
	PHT201A2_pHlevelR2 AT %IW0 : REAL;
	PHT201A2_pHlevelR2_ScaledValue:INT;
	PHT201A3_pHlevelR3 AT %IW0 : REAL;
	PHT201A3_pHlevelR3_ScaledValue:INT;
	PHT201A4_pHlevelR4 AT %IW0 : REAL;
	PHT201A4_pHlevelR4_ScaledValue:INT;
	XV205A_SBRValveR1_OpenCmd AT %Q* : BOOL;
	XV206A_SBRValveR2_OpenCmd AT %Q* : BOOL;
	XV207A_SBRValveR3_OpenCmd AT %Q* : BOOL;
	XV208A_SBRValveR4_OpenCmd AT %Q* : BOOL;
	XV201A_AirBlowerValveR1_OpenCmd AT %Q* : BOOL;
	XV202A_AirBlowerValveR2_OpenCmd AT %Q* : BOOL;
	XV203A_AirBlowerValveR3_OpenCmd AT %Q* : BOOL;
	XV204A_AirBlowerValveR4_OpenCmd AT %Q* : BOOL;
	XV221A_LimeValveR1_OpenCmd AT %Q* : BOOL;
	XV222A_LimeValveR2_OpenCmd AT %Q* : BOOL;
	XV223A_LimeValveR3_OpenCmd AT %Q* : BOOL;
	XV224A_LimeValveR4_OpenCmd AT %Q* : BOOL;
	XV211A_AlumValveR1_OpenCmd AT %Q* : BOOL;
	XV212A_AlumValveR2_OpenCmd AT %Q* : BOOL;
	XV213A_AlumValveR3_OpenCmd AT %Q* : BOOL;
	XV214A_AlumValveR4_OpenCmd AT %Q* : BOOL;
	XV241A_SludgeValveR1_OpenCmd AT %Q* : BOOL;
	XV242A_SludgeValveR2_OpenCmd AT %Q* : BOOL;
	XV243A_SludgeValveR3_OpenCmd AT %Q* : BOOL;
	XV244A_SludgeValveR4_OpenCmd AT %Q* : BOOL;
	XV241A_SludgeValveR1_CloseCmd AT %Q* : BOOL;
	XV242A_SludgeValveR2_CloseCmd AT %Q* : BOOL;
	XV243A_SludgeValveR3_CloseCmd AT %Q* : BOOL;
	XV244A_SludgeValveR4_CloseCmd AT %Q* : BOOL;
	XV205A_SBRValveR1_CloseCmd AT %Q* : BOOL;
	XV206A_SBRValveR2_CloseCmd AT %Q* : BOOL;
	XV207A_SBRValveR3_CloseCmd AT %Q* : BOOL;
	XV208A_SBRValveR4_CloseCmd AT %Q* : BOOL;
	XV201A_AirBlowerValveR1_CloseCmd AT %Q* : BOOL;
	XV202A_AirBlowerValveR2_CloseCmd AT %Q* : BOOL;
	XV203A_AirBlowerValveR3_CloseCmd AT %Q* : BOOL;
	XV204A_AirBlowerValveR4_CloseCmd AT %Q* : BOOL;
	XV221A_LimeValveR1_CloseCmd AT %Q* : BOOL;
	XV222A_LimeValveR2_CloseCmd AT %Q* : BOOL;
	XV223A_LimeValveR3_CloseCmd AT %Q* : BOOL;
	XV224A_LimeValveR4_CloseCmd AT %Q* : BOOL;
	XV211A_AlumValveR1_CloseCmd AT %Q* : BOOL;
	XV212A_AlumValveR2_CloseCmd AT %Q* : BOOL;
	XV213A_AlumValveR3_CloseCmd AT %Q* : BOOL;
	XV214A_AlumValveR4_CloseCmd AT %Q* : BOOL;
	OPR1AON_ReactorR1_OnlineCmd AT %Q* : BOOL;
	OPR2AON_ReactorR2_OnlineCmd AT %Q* : BOOL;
	OPR3AON_ReactorR3_OnlineCmd AT %Q* : BOOL;
	OPR4AON_ReactorR4_OnlineCmd AT %Q* : BOOL;
	OPR1AOFF_ReactorR1_OfflineCmd AT %Q* : BOOL;
	OPR2AOFF_ReactorR2_OfflineCmd AT %Q* : BOOL;
	OPR3AOFF_ReactorR3_OfflineCmd AT %Q* : BOOL;
	OPR4AOFF_ReactorR4_OfflineCmd AT %Q* : BOOL;
	OPR1ASW_ReactorR1_SwitchCmd AT %Q* : BOOL;
	OPR2ASW_ReactorR2_SwitchCmd AT %Q* : BOOL;
	OPR3ASW_ReactorR3_SwitchCmd AT %Q* : BOOL;
	OPR4ASW_ReactorR4_SwitchCmd AT %Q* : BOOL;
	AUX402_PLCRunStat AT %Q* : BOOL;
	AUX401_CommonAlarm AT %Q* : BOOL;
	LSH201B1_LevelSensorR1 AT %I* : BOOL;
	LSH201B2_LevelSensorR2 AT %I* : BOOL;
	LSH201B3_LevelSensorR3 AT %I* : BOOL;
	LSH201B4_LevelSensorR4 AT %I* : BOOL;
	OPR1B_ReactorStatus AT %I* : BOOL;
	OPR2B_ReactorStatus AT %I* : BOOL;
	OPR3B_ReactorStatus AT %I* : BOOL;
	OPR4B_ReactorStatus AT %I* : BOOL;
	DP05_DoorPanelStatus AT %I* : BOOL;
	TMT05_FanStatus AT %I* : BOOL;
	HR201B1_DecantHighLevelR1 AT %I* : BOOL;
	LR201B1_DecantLowLevelR1 AT %I* : BOOL;
	HR201B2_DecantHighLevelR2 AT %I* : BOOL;
	LR201B2_DecantLowLevelR2 AT %I* : BOOL;
	HR201B3_DecantHighLevelR3 AT %I* : BOOL;
	HR201B4_DecantHighLevelR4 AT %I* : BOOL;
	LR201B3_DecantLowLevelR3 AT %I* : BOOL;
	LR201B4_DecantLowLevelR4 AT %I* : BOOL;
	XV205B_SBRValveR1_OpenStat AT %I* : BOOL;
	XV206B_SBRValveR2_OpenStat AT %I* : BOOL;
	XV207B_SBRValveR3_OpenStat AT %I* : BOOL;
	XV208B_SBRValveR4_OpenStat AT %I* : BOOL;
	XV201B_AirBlowerValveR1_OpenStat AT %I* : BOOL;
	XV202B_AirBlowerValveR2_OpenStat AT %I* : BOOL;
	XV203B_AirBlowerValveR3_OpenStat AT %I* : BOOL;
	XV204B_AirBlowerValveR4_OpenStat AT %I* : BOOL;
	XV221B_LimeValveR1_OpenStat AT %I* : BOOL;
	XV222B_LimeValveR2_OpenStat AT %I* : BOOL;
	XV223B_LimeValveR3_OpenStat AT %I* : BOOL;
	XV224B_LimeValveR4_OpenStat AT %I* : BOOL;
	XV211B_AlumValveR1_OpenStat AT %I* : BOOL;
	XV212B_AlumValveR2_OpenStat AT %I* : BOOL;
	XV213B_AlumValveR3_OpenStat AT %I* : BOOL;
	XV214B_AlumValveR4_OpenStat AT %I* : BOOL;
	XV205B_SBRValveR1_CloseStat AT %I* : BOOL;
	XV206B_SBRValveR2_CloseStat AT %I* : BOOL;
	XV207B_SBRValveR3_CloseStat AT %I* : BOOL;
	XV208B_SBRValveR4_CloseStat AT %I* : BOOL;
	XV201B_AirBlowerValveR1_CloseStat AT %I* : BOOL;
	XV202B_AirBlowerValveR2_CloseStat AT %I* : BOOL;
	XV203B_AirBlowerValveR3_CloseStat AT %I* : BOOL;
	XV204B_AirBlowerValveR4_CloseStat AT %I* : BOOL;
	XV221B_LimeValveR1_CloseStat AT %I* : BOOL;
	XV222B_LimeValveR2_CloseStat AT %I* : BOOL;
	XV223B_LimeValveR3_CloseStat AT %I* : BOOL;
	XV224B_LimeValveR4_CloseStat AT %I* : BOOL;
	XV211B_AlumValveR1_CloseStat AT %I* : BOOL;
	XV212B_AlumValveR2_CloseStat AT %I* : BOOL;
	XV213B_AlumValveR3_CloseStat AT %I* : BOOL;
	XV214B_AlumValveR4_CloseStat AT %I* : BOOL;
	XV20xB_SludgeValveR1_CloseStat AT %I* : BOOL;
	XV20xB_SludgeValveR2_CloseStat AT %I* : BOOL;
	XV20xB_SludgeValveR3_CloseStat AT %I* : BOOL;
	XV20xB_SludgeValveR4_CloseStat AT %I* : BOOL;
	XV20xB_SludgeValveR1_OpenStat AT %I* : BOOL;
	XV20xB_SludgeValveR2_OpenStat AT %I* : BOOL;
	XV20xB_SludgeValveR3_OpenStat AT %I* : BOOL;
	XV20xB_SludgeValveR4_OpenStat AT %I* : BOOL;
	DO201B1_DOProfilesR1 AT %IW0 : REAL;
	DO201B1_DOProfilesR1_ScaledValue:INT;
	DO201B2_DOProfilesR2 AT %IW0 : REAL;
	DO201B2_DOProfilesR2_ScaledValue:INT;
	DO201B3_DOProfilesR3 AT %IW0 : REAL;
	DO201B3_DOProfilesR3_ScaledValue:INT;
	D0201B4_DOProfilesR4 AT %IW0 : REAL;
	D0201B4_DOProfilesR4_ScaledValue:INT;
	PHT201B1_pHlevelR1 AT %IW0 : REAL;
	PHT201B1_pHlevelR1_ScaledValue:INT;
	PHT201B2_pHlevelR2 AT %IW0 : REAL;
	PHT201B2_pHlevelR2_ScaledValue:INT;
	PHT201B3_pHlevelR3 AT %IW0 : REAL;
	PHT201B3_pHlevelR3_ScaledValue:INT;
	PHT201B4_pHlevelR4 AT %IW0 : REAL;
	PHT201B4_pHlevelR4_ScaledValue:INT;
	XV205B_SBRValveR1_OpenCmd AT %Q* : BOOL;
	XV206B_SBRValveR2_OpenCmd AT %Q* : BOOL;
	XV207B_SBRValveR3_OpenCmd AT %Q* : BOOL;
	XV208B_SBRValveR4_OpenCmd AT %Q* : BOOL;
	XV202B_AirBlowerValveR2_OpenCmd AT %Q* : BOOL;
	XV201B_AirBlowerValveR1_OpenCmd AT %Q* : BOOL;
	XV204B_AirBlowerValveR4_OpenCmd AT %Q* : BOOL;
	XV203B_AirBlowerValveR3_OpenCmd AT %Q* : BOOL;
	XV221B_LimeValveR1_OpenCmd AT %Q* : BOOL;
	XV222B_LimeValveR2_OpenCmd AT %Q* : BOOL;
	XV223B_LimeValveR3_OpenCmd AT %Q* : BOOL;
	XV224B_LimeValveR4_OpenCmd AT %Q* : BOOL;
	XV211B_AlumValveR1_OpenCmd AT %Q* : BOOL;
	XV212B_AlumValveR2_OpenCmd AT %Q* : BOOL;
	XV213B_AlumValveR3_OpenCmd AT %Q* : BOOL;
	XV214B_AlumValveR4_OpenCmd AT %Q* : BOOL;
	XV241B_SludgeValveR1_OpenCmd AT %Q* : BOOL;
	XV242B_SludgeValveR2_OpenCmd AT %Q* : BOOL;
	XV243B_SludgeValveR3_OpenCmd AT %Q* : BOOL;
	XV244B_SludgeValveR4_OpenCmd AT %Q* : BOOL;
	XV241B_SludgeValveR1_CloseCmd AT %Q* : BOOL;
	XV242B_SludgeValveR2_CloseCmd AT %Q* : BOOL;
	XV243B_SludgeValveClosedR3_CloseCmd AT %Q* : BOOL;
	XV244B_SludgeValveR4_CloseCmd AT %Q* : BOOL;
	XV205B_SBRValveR1_CloseCmd AT %Q* : BOOL;
	XV206B_SBRValveR2_CloseCmd AT %Q* : BOOL;
	XV207B_SBRValveR3_CloseCmd AT %Q* : BOOL;
	XV208B_SBRValveR4_CloseCmd AT %Q* : BOOL;
	XV201B_AirBlowerValveR1_CloseCmd AT %Q* : BOOL;
	XV202B_AirBlowerValveR2_CloseCmd AT %Q* : BOOL;
	XV203B_AirBlowerValveR3_CloseCmd AT %Q* : BOOL;
	XV204B_AirBlowerValveR4_CloseCmd AT %Q* : BOOL;
	XV221B_LimeValveR1_CloseCmd AT %Q* : BOOL;
	XV222B_LimeValveR2_CloseCmd AT %Q* : BOOL;
	XV223B_LimeValveR3_CloseCmd AT %Q* : BOOL;
	XV224B_LimeValveR4_CloseCmd AT %Q* : BOOL;
	XV211B_AlumValveR1_CloseCmd AT %Q* : BOOL;
	XV212B_AlumValveR2_CloseCmd AT %Q* : BOOL;
	XV213B_AlumValveR3_CloseCmd AT %Q* : BOOL;
	XV214B_AlumValveR4_CloseCmd AT %Q* : BOOL;
	OPR1BON_ReactorR1_OnlineCmd AT %Q* : BOOL;
	OPR2BON_ReactorR2_OnlineCmd AT %Q* : BOOL;
	OPR3BON_ReactorR3_OnlineCmd AT %Q* : BOOL;
	OPR4BON_ReactorR4_OnlineCmd AT %Q* : BOOL;
	OPR1BOFF_ReactorR1_OfflineCmd AT %Q* : BOOL;
	OPR2BOFF_ReactorR2_OfflineCmd AT %Q* : BOOL;
	OPR3BOFF_ReactorR3_OfflineCmd AT %Q* : BOOL;
	OPR4BOFF_ReactorR4_OfflineCmd AT %Q* : BOOL;
	OPR1BSW_ReactorR1_SwitchCmd AT %Q* : BOOL;
	OPR2BSW_ReactorR2_SwitchCmd AT %Q* : BOOL;
	OPR3BSW_ReactorR3_SwitchCmd AT %Q* : BOOL;
	OPR4BSW_ReactorR4_SwitchCmd AT %Q* : BOOL;
	AUX502_PLCRunStat AT %Q* : BOOL;
	AUX501_CommonAlarm AT %Q* : BOOL;
	LSHH210A_LimeTank1 AT %I* : BOOL;
	LSH210A_LimeTank1 AT %I* : BOOL;
	LSL210A_LimeTank1 AT %I* : BOOL;
	LSD210A_LimeTank1 AT %I* : BOOL;
	LSHH210B_LimeTank2 AT %I* : BOOL;
	LSH210B_LimeTank2 AT %I* : BOOL;
	LSL210B_LimeTank2 AT %I* : BOOL;
	LSD210B_LimeTank2 AT %I* : BOOL;
	LSHH210C_LimeTank3 AT %I* : BOOL;
	LSH210C_LimeTank3 AT %I* : BOOL;
	LSL210C_LimeTank3 AT %I* : BOOL;
	LSD210C_LimeTank3 AT %I* : BOOL;
	LSL351A_AlumTank1 AT %I* : BOOL;
	LSL351B_AlumTank2 AT %I* : BOOL;
	LSL351C_AlumTank3 AT %I* : BOOL;
	LSL351D_AlumTank4 AT %I* : BOOL;
	LSL355A_SodiumHypochloriteTank AT %I* : BOOL;
	LSL355B_SodiumHypochloriteTank AT %I* : BOOL;
	LSL355C_SodiumHypochloriteTank AT %I* : BOOL;
	LSL353A_CausticSodaTank AT %I* : BOOL;
	LSL353B_CausticSodaTank AT %I* : BOOL;
	LSHH301_EffluentSump AT %I* : BOOL;
	LSH301_EffluentSump AT %I* : BOOL;
	LSL301_EffluentSump AT %I* : BOOL;
	LSHH302_CollectionSump AT %I* : BOOL;
	LSH302_CollectionSump AT %I* : BOOL;
	LSL302_CollectionSump AT %I* : BOOL;
	LSH308A_ReUseWaterStorageTank1HIGH AT %I* : BOOL;
	LSH308B_ReUseWaterStorageTank2HIGH AT %I* : BOOL;
	XV251A_LimeSelectorTank_OpenStat AT %I* : BOOL;
	XV251B_LimeSelectorTank_OpenStat AT %I* : BOOL;
	XV251C_LimeSelectorTank_OpenStat AT %I* : BOOL;
	XV251A_LimeSelectorTank_CloseStat AT %I* : BOOL;
	XV251B_LimSelectorTank_CloseStat AT %I* : BOOL;
	XV251C_LimeSelectorTank_CloseStat AT %I* : BOOL;
	OPAlumA_AlumSelectorTank AT %I* : BOOL;
	OPAlumB_AlumSelectorTank AT %I* : BOOL;
	OPAlumC_AlumSelectorTank AT %I* : BOOL;
	OPAlumD_AlumSelectorTank AT %I* : BOOL;
	OPCausticA_CausticSodaSelectorTank1 AT %I* : BOOL;
	OPCausticB_CausticSodaSelectorTank2 AT %I* : BOOL;
	OPSodiumA_SodiumHypochloriteSelectorTank1 AT %I* : BOOL;
	OPSodiumB_SodiumHypochloriteSelectorTank2 AT %I* : BOOL;
	OPSodiumC_SodiumHypochloriteSelectorTank3 AT %I* : BOOL;
	P210A1_LimePumpS1_RunStat AT %I* : BOOL;
	P210A2_LimePumpS1S2_RunStat AT %I* : BOOL;
	P210A3_LimePumpS2_RunStat AT %I* : BOOL;
	P203A_LimeCirculationPump_RunStat AT %I* : BOOL;
	P203B_LimeCirculationPump_RunStat AT %I* : BOOL;
	P211A1_AlumPumpSBRS1_RunStat AT %I* : BOOL;
	P211A2_AlumPumpSBRS1_RunStat AT %I* : BOOL;
	P211B1_AlumPump1SBRS2_RunStat AT %I* : BOOL;
	P211B2_AlumPumpSBRS2_RunStat AT %I* : BOOL;
	P352A_AlumPumpTertiaryDosing_RunStat AT %I* : BOOL;
	P352B_AlumPumpTertiaryDosing_RunStat AT %I* : BOOL;
	XV210A1_LimeValveS1_OpenStat AT %I* : BOOL;
	XV201A2_LimeValveS2_OpenStat AT %I* : BOOL;
	XV210A1_LimeValveS1_CloseStat AT %I* : BOOL;
	XV201A2_LimeValveS2_CloseStat AT %I* : BOOL;
	P354A_CausticSodaPump_RunStat AT %I* : BOOL;
	P354B_CausticSodaPump_RunStat AT %I* : BOOL;
	P356A_SodiumHypochloritePumpChlorinetank_RunStat AT %I* : BOOL;
	P356B_SodiumHypochloritePumpChlorinetank_RunStat AT %I* : BOOL;
	P204A_SodiumHypochloritePumpDisinfectionTank_RunStat AT %I* : BOOL;
	P204B_SodiumHypochloritePumpDisinfectionTank_RunStat AT %I* : BOOL;
	M210A_LimeStirrer_OverloadStat AT %I* : BOOL;
	M210B_LimeStirrer_OverloadStat AT %I* : BOOL;
	M210C_LimeStirrer_OverloadStat AT %I* : BOOL;
	TMT06_FanStatus AT %I* : BOOL;
	DP06_DoorPanelStatus AT %I* : BOOL;
	XV250A_LimeWaterIntakeTank_OpenStat AT %I* : BOOL;
	XV250B_LimeWaterIntakeTank_OpenStat AT %I* : BOOL;
	XV250C_LimeWaterIntakeTank_OpenStat AT %I* : BOOL;
	XV250A_LimeWaterIntakeTank_CloseStat AT %I* : BOOL;
	XV250B_LimeWaterIntakeTank_CloseStat AT %I* : BOOL;
	XV250C_LimeWaterIntakeTank_CloseStat AT %I* : BOOL;
	XV303A_LamellaSludgeDischarge_OpenStat AT %I* : BOOL;
	XV303B_LamellaSludgeDischarge_OpenStat AT %I* : BOOL;
	XV303C_LamellaSludgeDischarge_OpenStat AT %I* : BOOL;
	XV303D_LamellaSludgeDischarge_OpenStat AT %I* : BOOL;
	XV305_TertiaryTreatmentMainValve_OpenStat AT %I* : BOOL;
	XV303A_LamellaSludgeDischarge_CloseStat AT %I* : BOOL;
	XV303B_LamellaSludgeDischarge_CloseStat AT %I* : BOOL;
	XV303C_LamellaSludgeDischarge_CloseStat AT %I* : BOOL;
	XV303D_LamellaSludgeDischarge_CloseStat AT %I* : BOOL;
	XV305_TertiaryTreatmentMainValve_CloseStat AT %I* : BOOL;
	M210A_LimeStirrer_RunStat AT %I* : BOOL;
	M210B_LimeStirrer_RunStat AT %I* : BOOL;
	M210C_LimeStirrer_RunStat AT %I* : BOOL;
	M303A_Floculator_RunStat AT %I* : BOOL;
	M303B_Floculator_RunStat AT %I* : BOOL;
	M303C_Floculator_RunStat AT %I* : BOOL;
	M303D_Floculator_RunStat AT %I* : BOOL;
	P301A_EffluentTransferPump_RunStat AT %I* : BOOL;
	P301B_EffluentTransferPump_RunStat AT %I* : BOOL;
	P302A_CollectionPump_RunStat AT %I* : BOOL;
	P302B_CollectionPump_RunStat AT %I* : BOOL;
	K301A_AirCompressor_RunStat AT %I* : BOOL;
	K301B_AirCompressor_RunStat AT %I* : BOOL;
	P210A1_LimePumpS1_LocalRemoteStat AT %I* : BOOL;
	P210A2_LimePumpS1_LocalRemoteStat AT %I* : BOOL;
	P210A3_LimePumpS1_LocalRemoteStat AT %I* : BOOL;
	P203A_LimeCirculationPump1_LocalRemoteStat AT %I* : BOOL;
	P203B_LimeCirculationPump2_LocalRemoteStat AT %I* : BOOL;
	P211A1_AlumPumpSBRS1_LocalRemoteStat AT %I* : BOOL;
	P211A2_AlumPumpSBRS1_LocalRemoteStat AT %I* : BOOL;
	P211B1_AlumPumpSBRS2_LocalRemoteStat AT %I* : BOOL;
	P211B2_AlumPump2SBRS2_LocalRemoteStat AT %I* : BOOL;
	P352A_AlumPumpTertiaryDosing_LocalRemoteStat AT %I* : BOOL;
	P352B_AlumPumpTertiaryDosing_LocalRemoteStat AT %I* : BOOL;
	P354A_CausticSodaPump_LocalRemoteStat AT %I* : BOOL;
	P354B_CausticSodaPump_LocalRemoteStat AT %I* : BOOL;
	P356A_SodiumHypochloritePump_LocalRemoteStat AT %I* : BOOL;
	P356B_SodiumHypochloritePump_LocalRemoteStat AT %I* : BOOL;
	P301A_EffluentTransferPump_LocalRemoteStat AT %I* : BOOL;
	P301B_EffluentTransferPump_LocalRemoteStat AT %I* : BOOL;
	P302A_CollectionPump_LocalRemoteStat AT %I* : BOOL;
	P302B_CollectionPump_LocalRemoteStat AT %I* : BOOL;
	K301A_AirCompressor_LocalRemoteStat AT %I* : BOOL;
	K301B_AirCompressor_LocalRemoteStat AT %I* : BOOL;
	M210A_LimeStirrer_LocalRemoteStat AT %I* : BOOL;
	M210B_LimeStirrer_LocalRemoteStat AT %I* : BOOL;
	M210C_LimeStirrer_LocalRemoteStat AT %I* : BOOL;
	P210A1_LimePumpS1_TripStat AT %I* : BOOL;
	P210A2_LimePumpS1_TripStat AT %I* : BOOL;
	P210A3_LimePumpS1_TripStat AT %I* : BOOL;
	P203A_LimeCirculationPump_TripStat AT %I* : BOOL;
	P203B_LimeCirculationPump_TripStat AT %I* : BOOL;
	P211A1_AlumPumpSBRS1_TripStat AT %I* : BOOL;
	P211A2_AlumPumpSBRS1_TripStat AT %I* : BOOL;
	P211B1_AlumPumpSBRS1_TripStat AT %I* : BOOL;
	P211B2_AlumPumpSBRS2_TripStat AT %I* : BOOL;
	P352A_AlumPumpTertiaryDosing_TripStat AT %I* : BOOL;
	P352B_AlumPumpTertiaryDosing_TripStat AT %I* : BOOL;
	P354A_CausticSodaPump_TripStat AT %I* : BOOL;
	P354B_CausticSodaPump_TripStat AT %I* : BOOL;
	P356A_SodiumHypochloritePump_TripStat AT %I* : BOOL;
	P356B_SodiumHypochloritePump_TripStat AT %I* : BOOL;
	P301A_EffluentTransferPump_TripStat AT %I* : BOOL;
	P301B_EffluentTransferPump_TripStat AT %I* : BOOL;
	P302A_CollectionPump_TripStat AT %I* : BOOL;
	P302B_CollectionPump_TripStat AT %I* : BOOL;
	K301A_AirCompressor_TripStat AT %I* : BOOL;
	K301B_AirCompressor_TripStat AT %I* : BOOL;
	M303A_Floculator_TripStat AT %I* : BOOL;
	M303B_Floculator_TripStat AT %I* : BOOL;
	M303C_Floculator_TripStat AT %I* : BOOL;
	M303D_Floculator_TripStat AT %I* : BOOL;
	P210A1_LimePumpS1_EStopStat AT %I* : BOOL;
	P210A2_LimePumpS1_EStopStat AT %I* : BOOL;
	P210A3_LimePumpS1_EStopStat AT %I* : BOOL;
	P203A_LimeCirculationPump_EStopStat AT %I* : BOOL;
	P203B_LimeCirculationPump_EStopStat AT %I* : BOOL;
	P211A1_AlumPumpSBRS1_EStopStat AT %I* : BOOL;
	P211A2_AlumPumpSBRS1_EStopStat AT %I* : BOOL;
	P211B1_AlumPumpSBRS2_EStopStat AT %I* : BOOL;
	P211B2_AlumPumpSBRS2_EStopStat AT %I* : BOOL;
	P352A_AlumPumpTertiaryDosing_EStopStat AT %I* : BOOL;
	P352B_AlumPumpTertiaryDosing_EStopStat AT %I* : BOOL;
	P354A_CausticSodaPump_EStopStat AT %I* : BOOL;
	P354B_CausticSodaPump_EStopStat AT %I* : BOOL;
	P356A_SodiumHypochloritePump_EStopStat AT %I* : BOOL;
	P356B_SodiumHypochloritePump_EStopStat AT %I* : BOOL;
	P301A_EffluentTransferPump_EStopStat AT %I* : BOOL;
	P301B_EffluentTransferPump_EStopStat AT %I* : BOOL;
	P302A_CollectionPump_EStopStat AT %I* : BOOL;
	P302B_CollectionPump_EStopStat AT %I* : BOOL;
	K301A_AirCompressor_EStopStat AT %I* : BOOL;
	K301B_AirCompressor_EStopStat AT %I* : BOOL;
	M210A_LimeStirrer_EStopStat AT %I* : BOOL;
	M210B_LimeStirrer_EStopStat AT %I* : BOOL;
	M210C_LimeStirrer_EStopStat AT %I* : BOOL;
	XV250A_LimeWaterIntakeTank_OpenCmd AT %Q* : BOOL;
	XV250B_LimeWaterIntakeTank_OpenCmd AT %Q* : BOOL;
	XV250C_LimeWaterIntakeTank_OpenCmd AT %Q* : BOOL;
	XV251A_LimeSelectorTank_OpenCmd AT %Q* : BOOL;
	XV251B_LimeSelectorTank_OpenCmd AT %Q* : BOOL;
	XV251C_LimeSelectorTank_OpenCmd AT %Q* : BOOL;
	M210A_LimeStirrer_RunCmd AT %Q* : BOOL;
	M210B_LimeStirrer_RunCmd AT %Q* : BOOL;
	M210C_LimeStirrer_RunCmd AT %Q* : BOOL;
	P210A1_LimePumpS1_RunCmd AT %Q* : BOOL;
	P210A2_LimePumpS1_RunCmd AT %Q* : BOOL;
	P210A3_LimePumpS1_RunCmd AT %Q* : BOOL;
	P210A1_LimeValveS2_OpenCmd AT %Q* : BOOL;
	P210A2_LimeValveS2_OpenCmd AT %Q* : BOOL;
	P354A_CausticSodaPump_RunCmd AT %Q* : BOOL;
	P354B_CausticSodaPump_RunCmd AT %Q* : BOOL;
	P356A_SodiumHypochloritePump_RunCmd AT %Q* : BOOL;
	P356B_SodiumHypochloritePump_RunCmd AT %Q* : BOOL;
	P204A_SodiumHypochloritePump_RunCmd AT %Q* : BOOL;
	P211A1_AlumPumpSBRS1_RunCmd AT %Q* : BOOL;
	P211A2_AlumPumpSBRS1_RunCmd AT %Q* : BOOL;
	P211B1_AlumPumpSBRS2_RunCmd AT %Q* : BOOL;
	P211B2_AlumPumpSBRS2_RunCmd AT %Q* : BOOL;
	P352A_AlumPumpTertiaryDosing_RunCmd AT %Q* : BOOL;
	P352B_AlumPumpTertiaryDosing_RunCmd AT %Q* : BOOL;
	P203A_LimeCirculationPump_RunCmd AT %Q* : BOOL;
	P203B_LimeCirculationPump_RunCmd AT %Q* : BOOL;
	XV303A_LamellaSludgeDischarge_RunCmd AT %Q* : BOOL;
	XV303B_LamellaSludgeDischarge_RunCmd AT %Q* : BOOL;
	XV303C_LamellaSludgeDischarge_RunCmd AT %Q* : BOOL;
	XV303D_LamellaSludgeDischarge_RunCmd AT %Q* : BOOL;
	XV305_TertiaryTreatmentMainValve_OpenCmd AT %Q* : BOOL;
	M303A_Floculator_RunCmd AT %Q* : BOOL;
	M303B_Floculator_RunCmd AT %Q* : BOOL;
	M303C_Floculator_RunCmd AT %Q* : BOOL;
	M303D_Floculator_RunCmd AT %Q* : BOOL;
	P301A_EffluentTransferPump_RunCmd AT %Q* : BOOL;
	P301B_EffluentTransferPump_RunCmd AT %Q* : BOOL;
	P302A_CollectionPump_RunCmd AT %Q* : BOOL;
	P302B_CollectionPump_RunCmd AT %Q* : BOOL;
	K301A_AirCompressor_RunCmd AT %Q* : BOOL;
	K301B_AirCompressor_RunCmd AT %Q* : BOOL;
	AUX1_CirculationOverflow AT %Q* : BOOL;
	AUX2_SystemInletMonitoring AT %Q* : BOOL;
	AUX3_SystemOutletMonitoring AT %Q* : BOOL;
	AUX4_ChlorineHIGH AT %Q* : BOOL;
	AUX5_SBRDosing AT %Q* : BOOL;
	AUX6_ChlorineDosing AT %Q* : BOOL;
	AUX7_DisinfectionDosing AT %Q* : BOOL;
	AUX8_TertiaryDosing AT %Q* : BOOL;
	AUX602_PLCRunStat AT %Q* : BOOL;
	AUX601_CommonAlarm AT %Q* : BOOL;
	AUX17_LimeInService AT %Q* : BOOL;
	AUX18_LimeInService AT %Q* : BOOL;
	AUX19_LimeInService AT %Q* : BOOL;
	AUX20_AlumInService AT %Q* : BOOL;
	AUX21_AlumInService AT %Q* : BOOL;
	AUX22_AlumInService AT %Q* : BOOL;
	AUX23_AlumInService AT %Q* : BOOL;
	AUX24_CausticInService AT %Q* : BOOL;
	AUX25_CausticInService AT %Q* : BOOL;
	AUX26_SodiumInService AT %Q* : BOOL;
	AUX27_SodiumInService AT %Q* : BOOL;
	AUX28_SodiumInService AT %Q* : BOOL;
	AUX33_LimeLOW AT %Q* : BOOL;
	AUX34_LimeLOW AT %Q* : BOOL;
	AUX35_LimeLOW AT %Q* : BOOL;
	AUX36_AlumLOW AT %Q* : BOOL;
	AUX37_AlumLOW AT %Q* : BOOL;
	AUX38_AlumLOW AT %Q* : BOOL;
	AUX39_AlumLOW AT %Q* : BOOL;
	AUX40_CausticLOW AT %Q* : BOOL;
	AUX41_CausticLOW AT %Q* : BOOL;
	AUX42_SodiumLOW AT %Q* : BOOL;
	AUX43_SodiumLOW AT %Q* : BOOL;
	AUX44_SodiumLOW AT %Q* : BOOL;
	FT300_EffluentFlowrateEntry AT %IW0 : REAL;
	FT300_EffluentFlowrateEntry_ScaledValue:INT;
	AT300_EffluentTurbidityEntry AT %IW0 : REAL;
	AT300_EffluentTurbidityEntry_ScaledValue:INT;
	PHT301_EffluentpHLevelEntry AT %IW0 : REAL;
	PHT301_EffluentpHLevelEntry_ScaledValue:INT;
	FT301_TreatedEffluentFlowrateDischarge AT %IW0 : REAL;
	FT301_TreatedEffluentFlowrateDischarge_ScaledValue:INT;
	AT302_TreatedEffluentTurbidityDischarge AT %IW0 : REAL;
	AT302_TreatedEffluentTurbidityDischarge_ScaledValue : INT;
	PHT303_TreatedEffluentpHLevelDischarge AT %IW0 : REAL;
	PHT303_TreatedEffluentpHLevelDischarge_ScaledValue:INT;
	CL303_ResidualChlorineAnalyzer AT %IW0 : REAL;
	CL303_ResidualChlorineAnalyzer_ScaledValue:INT;
	CL304_FinalChlorineAnalyzer AT %IW0 : REAL;
	CL304_FinalChlorineAnalyzer_ScaledValue:INT;
	ORP_DisinfectionTankAnalyzer AT %IW0 : REAL;
	ORP_DisinfectionTankAnalyzer_ScaledValue:INT;
	TMT07_FanStatus AT %I* : BOOL;
	DP07_DoorPanel AT %I* : BOOL;
	LSH501A_SludgeStorage AT %I* : BOOL;
	LSHH501A_SludgeStorage AT %I* : BOOL;
	LSL501A_SludgeStorage AT %I* : BOOL;
	LSH501B_SludgeStorage AT %I* : BOOL;
	LSHH501B_SludgeStorage AT %I* : BOOL;
	LSL501B_SludgeStorage AT %I* : BOOL;
	LSH620_FiltrateSumpLevel AT %I* : BOOL;
	LSL620_FiltrateSumpLevel AT %I* : BOOL;
	LSHPU501_PolymerTankLevel AT %I* : BOOL;
	LSLPU501_PolymerTankLevel AT %I* : BOOL;
	PSL505A_PressureSWWaterLine AT %I* : BOOL;
	PSL505B_PressureSWWaterLine2 AT %I* : BOOL;
	P501A_SludgeFeedPump_RunStat AT %I* : BOOL;
	P501B_SludgeFeedPump_RunStat AT %I* : BOOL;
	P501C_SludgeFeedPump_RunStat AT %I* : BOOL;
	B501A_Blower_RunStat AT %I* : BOOL;
	B501B_Blower_RunStat AT %I* : BOOL;
	B501C_Blower_RunStat AT %I* : BOOL;
	M502A_Floculator_RunStat AT %I* : BOOL;
	M502B_Floculator_RunStat AT %I* : BOOL;
	P602A_FiltratePump_RunStat AT %I* : BOOL;
	P602B_FiltratePump_RunStat AT %I* : BOOL;
	XV505A_SolenoidValveLine_OpenStat AT %I* : BOOL;
	XV505B_SolenoidValveLine_OpenStat AT %I* : BOOL;
	XVPU502_DiagpharmAirValve_OpenStat AT %I* : BOOL;
	XV505A_SolenoidValveLine_CloseStat AT %I* : BOOL;
	XV505B_SolenoidValveLine_CloseStat AT %I* : BOOL;
	XVPU502_DiagpharmAirValve_CloseStat AT %I* : BOOL;
	D503A_DrumThickener_RunStat AT %I* : BOOL;
	D503B_DrumThickener_RunStat AT %I* : BOOL;
	P505A_BackwashWaterPump_RunStat AT %I* : BOOL;
	P505B_BackwashWaterPump_RunStat AT %I* : BOOL;
	P505C_BackwashWaterPump_RunStat AT %I* : BOOL;
	XV501A_AirBlowerValve_OpenStat AT %I* : BOOL;
	XV501A_AirBlowerValve_CloseStat AT %I* : BOOL;
	XV501B_AirBlowerValve_OpenStat AT %I* : BOOL;
	XV501B_AirBlowerValve_CloseStat AT %I* : BOOL;
	XVPU501A_PolymerValve_OpenStat AT %I* : BOOL;
	XVPU501A_PolymerValve_CloseStat AT %I* : BOOL;
	XVPU501B_PolymerValve_OpenStat AT %I* : BOOL;
	XVPU501B_PolymerValve_ClosedStat AT %I* : BOOL;
	M503_PolymerStirrer_RunStat AT %I* : BOOL;
	XVW501A_WaterValve_OpenStat AT %I* : BOOL;
	XVW501A_WaterValve_CloseStat AT %I* : BOOL;
	B501A_Blower_OverloadStat AT %I* : BOOL;
	B501A_Blower_IncompleteStat AT %I* : BOOL;
	B501B_Blower_OverloadStat AT %I* : BOOL;
	B501B_Blower_IncompleteStat AT %I* : BOOL;
	B501C_Blower_OverloadStat AT %I* : BOOL;
	B501C_Blower_IncompleteStat AT %I* : BOOL;
	P501A_SludgeFeedPump_OverloadStat AT %I* : BOOL;
	P501A_SludgeFeedPump_IncompleteStat AT %I* : BOOL;
	P501B_SludgeFeedPump_OverloadStat AT %I* : BOOL;
	P501B_SludgeFeedPump_IncompleteStat AT %I* : BOOL;
	P501C_SludgeFeedPumpOverloadStat AT %I* : BOOL;
	P501C_SludgeFeedPump_IncompleteStat AT %I* : BOOL;
	P602A_FiltratePump_TripStat AT %I* : BOOL;
	P602B_FiltratePump_TripStat AT %I* : BOOL;
	M502A_Floculator_OverloadStat AT %I* : BOOL;
	M502B_Floculator_OverloadStat AT %I* : BOOL;
	D503A_DrumThickener_OverloadStat AT %I* : BOOL;
	D503B_DrumThickener_OverloadStat AT %I* : BOOL;
	P505A_BackwashWaterPump_OverloadStat AT %I* : BOOL;
	P505A_BackwashWaterPump_IncompleteStat AT %I* : BOOL;
	P505B_BackwashWaterPump_OverloadStat AT %I* : BOOL;
	P505B_BackwashWaterPump_IncompleteStat AT %I* : BOOL;
	P505C_BackwashWaterPump_OverloadStat AT %I* : BOOL;
	P505C_BackwashWaterPump_IncompleteStat AT %I* : BOOL;
	M503_PolymerStirrer_OverloadStat AT %I* : BOOL;
	P501A_SludgeFeedPump_LocalRemoteStat AT %I* : BOOL;
	P501B_SludgeFeedPump_LocalRemoteStat AT %I* : BOOL;
	P501C_SludgeFeedPump_LocalRemoteStat AT %I* : BOOL;
	B501A_Blower_LocalRemoteStat AT %I* : BOOL;
	B501B_Blower_LocalRemoteStat AT %I* : BOOL;
	B501C_Blower_LocalRemoteStat AT %I* : BOOL;
	M502A_Floculator_LocalRemoteStat AT %I* : BOOL;
	M502B_Floculator_LocalRemoteStat AT %I* : BOOL;
	D503A_DrumThickener_LocalRemoteStat AT %I* : BOOL;
	D503B_DrumThickener_LocalRemoteStat AT %I* : BOOL;
	P505A_BackwashWaterPump_LocalRemoteStat AT %I* : BOOL;
	P505B_BackwashWaterPump_LocalRemoteStat AT %I* : BOOL;
	P505C_BackwashWaterPump_LocalRemoteStat AT %I* : BOOL;
	P602A_FiltratePump_LocalRemoteStat AT %I* : BOOL;
	P602B_FiltratePump_LocalRemoteStat AT %I* : BOOL;
	M503_PolymerStirrer_LocalRemoteStat AT %I* : BOOL;
	P501A_SludgeFeedPump_EStopStat AT %I* : BOOL;
	P501B_SludgeFeedPump_EStopStat AT %I* : BOOL;
	P501C_SludgeFeedPump_EStopStat AT %I* : BOOL;
	B501A_Blower_EStopStat AT %I* : BOOL;
	B501B_Blower_EStopStat AT %I* : BOOL;
	B501C_Blower_EStopStat AT %I* : BOOL;
	M502A_Floculator_EStopStat AT %I* : BOOL;
	M502B_Floculator_EStopStat AT %I* : BOOL;
	D503A_DrumThickener_EStopStat AT %I* : BOOL;
	D503B_DrumThickener_EStopStat AT %I* : BOOL;
	P505A_BackwashWaterPump_EStopStat AT %I* : BOOL;
	P505B_BackwashWaterPump_EStopStat AT %I* : BOOL;
	P505C_BackwashWaterPump_EStopStat AT %I* : BOOL;
	P602A_FiltratePump_EStopStat AT %I* : BOOL;
	P602B_FiltratePump_EStopStat AT %I* : BOOL;
	M503_PolymerStirrer_EStopStat AT %I* : BOOL;
	VE801B_SuctionFan_OnOffStat AT %I* : BOOL;
	P802B_CirculationPump_OnOffStat AT %I* : BOOL;
	P803B_CirculationPump_OnOffStat AT %I* : BOOL;
	P804B_CirculationPump_OnOffStat AT %I* : BOOL;
	P805B1_H2S04Pump_OnOffStat AT %I* : BOOL;
	P805B2_H2S04Pump_OnOffStat AT %I* : BOOL;
	P806B1_NAOHPump_OnOffStat AT %I* : BOOL;
	P806B2_NAOHPump_OnOffStat AT %I* : BOOL;
	P807B1_NAOCLPump_OnOffStat AT %I* : BOOL;
	P807B2_NAOCLPump_OnOffStat AT %I* : BOOL;
	VE801B_SuctionFan_OverloadStat AT %I* : BOOL;
	P802B_CirculationPump_OverloadStat AT %I* : BOOL;
	P803B_CirculationPump_OverloadStat AT %I* : BOOL;
	P804B_CirculationPump_OverloadStat AT %I* : BOOL;
	P805B1_H2S04Pump_OverloadStat AT %I* : BOOL;
	P805B2_H2S04Pump_OverloadStat AT %I* : BOOL;
	P806B1_NAOHPump_OverloadStat AT %I* : BOOL;
	P806B2_NAOHPump_OverloadStat AT %I* : BOOL;
	P807B1_NAOCLPump_OverloadStat AT %I* : BOOL;
	P807B2_NAOCLPump_OverloadStat AT %I* : BOOL;
	VE801B_Suction_EStopStat AT %I* : BOOL;
	P802B_CirculationPump_EStopStat AT %I* : BOOL;
	P803B_CirculationPump_EStopStat AT %I* : BOOL;
	P804B_CirculationPump_EStopStat AT %I* : BOOL;
	P805B1_H2S04Pump_EStopStat AT %I* : BOOL;
	P805B2_H2S04Pump_EStopStat AT %I* : BOOL;
	P806B1_NAOHPump_EStopStat AT %I* : BOOL;
	P806B2_NAOHPump_EstopStat AT %I* : BOOL;
	P807B1_NAOCLPump_EStopStat AT %I* : BOOL;
	P807B2_NAOCLPump_EStopStat AT %I* : BOOL;
	LSH600_SludgePitSensor AT %IW0 : REAL;
	LSH600_SludgePitSensor_ScaledValue:INT;
	XVPU502_DiagpharmAirValve_OpenCmd AT %Q* : BOOL;
	M502A_Floculator_RunCmd AT %Q* : BOOL;
	M502B_Floculator_RunCmd AT %Q* : BOOL;
	M503A_DrumThickener_RunCmd AT %Q* : BOOL;
	M503B_DrumThickener_RunCmd AT %Q* : BOOL;
	P602A_FiltratePump_RunCmd AT %Q* : BOOL;
	P602B_FiltratePump_RunCmd AT %Q* : BOOL;
	XVPU501A_PolymerValve_OpenCmd AT %Q* : BOOL;
	XVPU501A_PolymerValve_CloseCmd AT %Q* : BOOL;
	XV505A_SolenoidValveLine_OpenCmd AT %Q* : BOOL;
	XV505B_SolenoidValveLine_CloseCmd AT %Q* : BOOL;
	XVW501A_WaterValve_OpenCmd AT %Q* : BOOL;
	B501A_Blower_RunCmd AT %Q* : BOOL;
	B501B_Blower_RunCmd AT %Q* : BOOL;
	B501C_Blower_RunCmd AT %Q* : BOOL;
	P501A_SludgeFeedPump_RunCmd AT %Q* : BOOL;
	P501B_SludgeFeedPump_RunCmd AT %Q* : BOOL;
	P501C_SludgeFeedPump_RunCmd AT %Q* : BOOL;
	P505A_BackwashWaterPump_RunCmd AT %Q* : BOOL;
	P505B_BackwashWaterPump_RunCmd AT %Q* : BOOL;
	P505C_BackwashWaterPump_RunCmd AT %Q* : BOOL;
	XV501A_AirBlowerValve_OpenCmd AT %Q* : BOOL;
	XV501B_AirBlowerValve_OpenCmd AT %Q* : BOOL;
	XV501A_AirBlowerValve_CloseCmd AT %Q* : BOOL;
	XV501B_AirBlowerValve_CloseCmd AT %Q* : BOOL;
	M503_PolymerStirrer_FwdCmd AT %Q* : BOOL;
	M503_PolymerStirrer_RvsCmd AT %Q* : BOOL;
	AUX510_SludgeStorageHigh AT %Q* : BOOL;
	AUX511_ReuseWaterStorageLow AT %Q* : BOOL;
	AUX512_FiltrateSumpHigh AT %Q* : BOOL;
	AUX513_SludgePitHigh AT %Q* : BOOL;
	AUX514_PolymerLevelLow AT %Q* : BOOL;
	AUX701_CommonAlarm AT %Q* : BOOL;
	AUX702_PLCRunStat AT %Q* : BOOL;
	LSL309A_WaterLevelTank AT %I* : BOOL;
	LSL309B_WaterLevelTank AT %I* : BOOL;
	LSH405_VacuumChestLevel AT %I* : BOOL;
	TMT08_FanStatus AT %I* : BOOL;
	DP08_DoorStatus AT %I* : BOOL;
	FSL101_FreshWaterActivationStatus AT %I* : BOOL;
	PSL412_PressureSwitch AT %I* : BOOL;
	PG413_LowPressureGauge AT %I* : BOOL;
	PG414_HighPressureGauge AT %I* : BOOL;
	XV401_SolenoidValve_OpenStat AT %I* : BOOL;
	XV401_SolenoidValve_CloseStat AT %I* : BOOL;
	P401A_LeadPumpA_OverloadStat AT %I* : BOOL;
	P401A_LeadPumpA_IncompleteStat AT %I* : BOOL;
	P401B_LeadPumpB_OverloadStat AT %I* : BOOL;
	P401B_LeadPumpB_IncompleteStat AT %I* : BOOL;
	P401C_LeadPumpC_OverloadStat AT %I* : BOOL;
	P401C_LeadPumpC_IncompleteStat AT %I* : BOOL;
	P401D_LeadPumpD_OverloadStat AT %I* : BOOL;
	P401D_LeadPumpD_IncompleteStat AT %I* : BOOL;
	P402A_JockeyPumpA_OverloadStat AT %I* : BOOL;
	P402A_JockeyPumpA_IncompleteStat AT %I* : BOOL;
	P402B_JockeyPumpB_OverloadStat AT %I* : BOOL;
	P402B_JockeyPumpB_IncompleteStat AT %I* : BOOL;
	P403A_VacuumPumpA_OverloadStat AT %I* : BOOL;
	P403B_VacuumPumpB_OverloadStat AT %I* : BOOL;
	P401A_LeadPumpA_LocalRemoteStat AT %I* : BOOL;
	P401B_LeadPumpB_LocalRemoteStat AT %I* : BOOL;
	P401C_LeadPumpC_LocalRemoteStat AT %I* : BOOL;
	P401D_LeadPumpD_LocalRemoteStat AT %I* : BOOL;
	P402A_JockeyPumpA_LocalRemoteStat AT %I* : BOOL;
	P402B_JockeyPumpB_LocalRemoteStat AT %I* : BOOL;
	P403A_VacuumPumpA_LocalRemoteStat AT %I* : BOOL;
	P403B_VacuumPumpB_LocalRemoteStat AT %I* : BOOL;
	P401A_LeadPumpA_OnOffStat AT %I* : BOOL;
	P401B_LeadPumpB_OnOffStat AT %I* : BOOL;
	P401C_LeadPumpC_OnOffStat AT %I* : BOOL;
	P401D_LeadPumpD_OnOffStat AT %I* : BOOL;
	P402A_JockeyPumpA_OnOffStat AT %I* : BOOL;
	P402B_JockeyPumpB_OnOffStat AT %I* : BOOL;
	P403A_VacuumPumpA_OnOffStat AT %I* : BOOL;
	P403B_VacuumPumpB_OnOffStat AT %I* : BOOL;
	P401A_LeadPumpA_EStopStat AT %I* : BOOL;
	P401B_LeadPumpB_EStopStat AT %I* : BOOL;
	P401C_LeadPumpC_EStopStat AT %I* : BOOL;
	P401D_LeadPumpD_EStopStat AT %I* : BOOL;
	P402A_JockeyPumpA_EStopStat AT %I* : BOOL;
	P402B_JockeyPumpB_EStopStat AT %I* : BOOL;
	P403A_VacuumPumpA_EStopStat AT %I* : BOOL;
	P403B_VacuumPumpB_EStopStat AT %I* : BOOL;
	XV401_SolenoidValve_OpenCmd AT %Q* : BOOL;
	P401A_LeadPumpA_RunCmd AT %Q* : BOOL;
	P401B_LeadPumpB_RunCmd AT %Q* : BOOL;
	P401C_LeadPumpC_RunCmd AT %Q* : BOOL;
	P401D_LeadPumpD_RunCmd AT %Q* : BOOL;
	P402A_JockeyPumpA_RunCmd AT %Q* : BOOL;
	P402B_JockeyPumpB_RunCmd AT %Q* : BOOL;
	P403A_VacuumPumpA_RunCmd AT %Q* : BOOL;
	P403B_VacuumPumpB_RunCmd AT %Q* : BOOL;
	AUX415_AuxLamp_LowPressure AT %Q* : BOOL;
	AUX416_AuxLamp_TankHighLevel AT %Q* : BOOL;
	AUX417_AuxLamp_SystemPrimed AT %Q* : BOOL;
	AUX801_CommonAlarm AT %Q* : BOOL;
	AUX802_PLCRunStatus AT %Q* : BOOL;
	PSL411_PressureTransmitter AT %IW0 : REAL;
	PSL411_PressureTransmitter_ScaledValue:INT;
	F900_FanStatus AT %I* : BOOL;
	D900_DoorPanelStat AT %I* : BOOL;
	GENRUN_Generator_RunStat AT %I* : BOOL;
	GENOT_Generator_OverloadStat AT %I* : BOOL;
	GENFAIL_Generator_FailStat AT %I* : BOOL;
	AUX902_PLCRunStatus AT %Q* : BOOL;
	AUX901_CommonAlarm AT %Q* : BOOL;
	AUX903_GeneratorSupplyStat AT %Q* : BOOL;
	AUX904_Stream1_RunStat AT %Q* : BOOL;
	AUX905_Stream2_RunStat AT %Q* : BOOL;
	AUX906_InletWork1_RunStat AT %Q* : BOOL;
	AUX907_BlowerHouse1_RunStat AT %Q* : BOOL;
	AUX908_SBR1_RunStat AT %Q* : BOOL;
	AUX909_InletWork2_RunStat AT %Q* : BOOL;
	AUX910_BlowerHouse2_RunStat AT %Q* : BOOL;
	AUX911_SBR2_RunStat AT %Q* : BOOL;
	AUX912_ChemicalTertiary_RunStat AT %Q* : BOOL;
	AUX913_SludgeThickening_RunStat AT %Q* : BOOL;
	AUX914_FilterPress_RunStat AT %Q* : BOOL;
	AUX915_Reuse_RunStat AT %Q* : BOOL;

(*Koupler Status*)
	ScadaRoom_KouplerUTP_State AT %I*:UINT;
	ScadaRoom_KouplerFiber_State AT %I*:UINT;
	InletWork_1_KouplerFiber_State AT %I*:UINT;
	InletWork_2_KouplerFiber_State AT %I*:UINT;
	BlowerHouse_2_KouplerFiber_State AT %I*:UINT;
	BlowerHouse_1_KouplerFiber_State AT %I*:UINT;
	SBR_1_KouplerFiber_State AT %I*:UINT;
	SBR_2_KouplerFiber_State AT %I*:UINT;
	ChemicalAndTertiary_KouplerFiber_State AT %I*:UINT;
	SludgeThickening_KouplerFiber_State AT %I*:UINT;
	Reused_KouplerFiber_State AT %I*:UINT;
	ScadaRoom_KouplerFiber_Return_State AT %I*:UINT;

	ScadaRoom_KouplerUTP_StateBool:BOOL;
	ScadaRoom_KouplerFiber_StateBool:BOOL;
	InletWork_1_KouplerFiber_StateBool:BOOL;
	InletWork_2_KouplerFiber_StateBool:BOOL;
	BlowerHouse_2_KouplerFiber_StateBool:BOOL;
	BlowerHouse_1_KouplerFiber_StateBool:BOOL;
	SBR_1_KouplerFiber_StateBool:BOOL;
	SBR_2_KouplerFiber_StateBool:BOOL;
	ChemicalAndTertiary_KouplerFiber_StateBool:BOOL;
	SludgeThickening_KouplerFiber_StateBool:BOOL;
	Reused_KouplerFiber_StateBool:BOOL;
	ScadaRoom_KouplerFiber_Return_StateBool:BOOL;

(*inlet*)
	INLET_A: INLET;
	rA1: BOOL;
	EQUIP_TYPE_1_EQA: EQUP_TYPE_1;
	r_eqA1: BOOL;
	EQUIP_TYPE_2_MXA: EQUIP_TYPE_2;
	EQUIP_TYPE_3_PSA1: EQUIP_TYPE_3;
	EQUIP_TYPE_3_PSA2: EQUIP_TYPE_3;
	EQUIP_TYPE_4_SCA: EQUIP_TYPE_4;
	EQUIP_TYPE_4_SPA: EQUIP_TYPE_4;
	EQUIP_TYPE_5_CWSA: EQUIP_TYPE_5;
	EQUIP_TYPE_4_FSA1: EQUIP_TYPE_4;
	EQUIP_TYPE_4_FSA2: EQUIP_TYPE_4;
	EQUIP_TYPE_6_WSA1: EQUIP_TYPE_6;
	EQUIP_TYPE_6_WSA2: EQUIP_TYPE_6;
	EQUIP_TYPE_5_GRVA1: EQUIP_TYPE_5;
	EQUIP_TYPE_5_GRVA2: EQUIP_TYPE_5;
	EQUIP_TYPE_4_ClassifierA: EQUIP_TYPE_4;
	EQUP_TYPE_1_STA1: EQUP_TYPE_1;
	r_STA1: BOOL;


	INLET_B: INLET;
	rB1: BOOL;
	EQUIP_TYPE_1_EQB: EQUP_TYPE_1;
	r_eqB1: BOOL;
	EQUIP_TYPE_2_MXB: EQUIP_TYPE_2;
	EQUIP_TYPE_3_PSB1: EQUIP_TYPE_3;
	EQUIP_TYPE_3_PSB2: EQUIP_TYPE_3;
	EQUIP_TYPE_4_SCB: EQUIP_TYPE_4;
	EQUIP_TYPE_4_SPB: EQUIP_TYPE_4;
	EQUIP_TYPE_5_CWSB: EQUIP_TYPE_5;
	EQUIP_TYPE_4_FSB1: EQUIP_TYPE_4;
	EQUIP_TYPE_4_FSB2: EQUIP_TYPE_4;
	EQUIP_TYPE_6_WSB1: EQUIP_TYPE_6;
	EQUIP_TYPE_6_WSB2: EQUIP_TYPE_6;
	EQUIP_TYPE_5_GRVB1: EQUIP_TYPE_5;
	EQUIP_TYPE_5_GRVB2: EQUIP_TYPE_5;
	EQUIP_TYPE_4_ClassifierB: EQUIP_TYPE_4;
	EQUP_TYPE_1_STB1: EQUP_TYPE_1;
	r_STB1: BOOL;

(*inlet blower*)
	EQUP_TYPE_7_Blower: EQUP_TYPE_7;
	rblower: BOOL;
(*CHEMICAL*)
	CHEMICAL_A: Chemical_new;

	reset_lime_tank_1: BOOL;
	reset_lime_tank_2: BOOL;
	reset_lime_tank_3: BOOL;

(*SBRA*)
	reactorA1: Reactor;
	resumeAlumA1: BOOL;
	Alum_reactorA1: TIME;

	reactorA2: Reactor;
	resumealumA2: BOOL;
	alum_reactorA2: TIME;

	reactorA3: Reactor;
	resumealumA3: BOOL;
	alum_reactorA3: TIME;

	reactorA4: Reactor;
	resumealumA4: BOOL;
	alum_reactorA4: TIME;


	fill_selectorA: Fill_selector;
	aerate_selectorA: blower_selector;
	decant_selectorA: Decant_selector;

	EQUIP_TYPE_3_Valva1_RA1: EQUIP_TYPE_9;
	EQUIP_TYPE_8_MIXER_A1: EQUIP_TYPE_8;
	EQUIP_TYPE_3_Valve2_RA1: EQUIP_TYPE_9;
	EQUIP_TYPE_3_Valve3_RA1: EQUIP_TYPE_9;
	EQUIP_TYPE_3_Valve4_RA1: EQUIP_TYPE_9;
	EQUIP_TYPE_9_Valve5_RA1: EQUIP_TYPE_9;
	EQUIP_TYPE_10_Dec_RA1: EQUIP_TYPE_10;
	reset_dec_RA1: BOOL;


	EQUIP_TYPE_3_Valva1_RA2: EQUIP_TYPE_9;
	EQUIP_TYPE_8_MIXER_A2: EQUIP_TYPE_8;
	EQUIP_TYPE_3_Valve2_RA2: EQUIP_TYPE_9;
	EQUIP_TYPE_3_Valve3_RA2: EQUIP_TYPE_9;
	EQUIP_TYPE_3_Valve4_RA2: EQUIP_TYPE_9;
	EQUIP_TYPE_9_Valve5_RA2: EQUIP_TYPE_9;
	EQUIP_TYPE_10_Dec_RA2: EQUIP_TYPE_10;
	reset_dec_RA2: BOOL;


	EQUIP_TYPE_3_Valva1_RA3: EQUIP_TYPE_9;
	EQUIP_TYPE_8_MIXER_A3: EQUIP_TYPE_8;
	EQUIP_TYPE_3_Valve2_RA3: EQUIP_TYPE_9;
	EQUIP_TYPE_3_Valve3_RA3: EQUIP_TYPE_9;
	EQUIP_TYPE_3_Valve4_RA3: EQUIP_TYPE_9;
	EQUIP_TYPE_9_Valve5_RA3: EQUIP_TYPE_9;
	EQUIP_TYPE_10_Dec_RA3: EQUIP_TYPE_10;
	reset_dec_RA3: BOOL;


	EQUIP_TYPE_3_Valva1_RA4: EQUIP_TYPE_9;
	EQUIP_TYPE_8_MIXER_A4: EQUIP_TYPE_8;
	EQUIP_TYPE_3_Valve2_RA4: EQUIP_TYPE_9;
	EQUIP_TYPE_3_Valve3_RA4: EQUIP_TYPE_9;
	EQUIP_TYPE_3_Valve4_RA4: EQUIP_TYPE_9;
	EQUIP_TYPE_9_Valve5_RA4: EQUIP_TYPE_9;
	EQUIP_TYPE_10_Dec_RA4: EQUIP_TYPE_10;
	reset_dec_RA4: BOOL;

	EQUP_TYPE_1_Pump_RA: EQUP_TYPE_1;
	reset_Pump2_RA: BOOL;

(*SBRB*)
	reactorB1: Reactor;
	resumeAlumB1: BOOL;
	Alum_reactorB1: TIME;

	reactorB2: Reactor;
	resumealumB2: BOOL;
	alum_reactorB2: TIME;

	reactorB3: Reactor;
	resumealumB3: BOOL;
	alum_reactorB3: TIME;

	reactorB4: Reactor;
	resumealumB4: BOOL;
	alum_reactorB4: TIME;


	fill_selectorB: Fill_selector;
	aerate_selectorB: blower_selector;
	decant_selectorB: Decant_selector;

	EQUIP_TYPE_3_Valva1_RB1: EQUIP_TYPE_9;
	EQUIP_TYPE_8_MIXER_B1: EQUIP_TYPE_8;
	EQUIP_TYPE_3_Valve2_RB1: EQUIP_TYPE_9;
	EQUIP_TYPE_3_Valve3_RB1: EQUIP_TYPE_9;
	EQUIP_TYPE_3_Valve4_RB1: EQUIP_TYPE_9;
	EQUIP_TYPE_9_Valve5_RB1: EQUIP_TYPE_9;
	EQUIP_TYPE_10_Dec_RB1: EQUIP_TYPE_10;
	reset_dec_RB1: BOOL;


	EQUIP_TYPE_3_Valva1_RB2: EQUIP_TYPE_9;
	EQUIP_TYPE_8_MIXER_B2: EQUIP_TYPE_8;
	EQUIP_TYPE_3_Valve2_RB2: EQUIP_TYPE_9;
	EQUIP_TYPE_3_Valve3_RB2: EQUIP_TYPE_9;
	EQUIP_TYPE_3_Valve4_RB2: EQUIP_TYPE_9;
	EQUIP_TYPE_9_Valve5_RB2: EQUIP_TYPE_9;
	EQUIP_TYPE_10_Dec_RB2: EQUIP_TYPE_10;
	reset_dec_RB2: BOOL;


	EQUIP_TYPE_3_Valva1_RB3: EQUIP_TYPE_9;
	EQUIP_TYPE_8_MIXER_B3: EQUIP_TYPE_8;
	EQUIP_TYPE_3_Valve2_RB3: EQUIP_TYPE_9;
	EQUIP_TYPE_3_Valve3_RB3: EQUIP_TYPE_9;
	EQUIP_TYPE_3_Valve4_RB3: EQUIP_TYPE_9;
	EQUIP_TYPE_9_Valve5_RB3: EQUIP_TYPE_9;
	EQUIP_TYPE_10_Dec_RB3: EQUIP_TYPE_10;
	reset_dec_RB3: BOOL;


	EQUIP_TYPE_3_Valva1_RB4: EQUIP_TYPE_9;
	EQUIP_TYPE_8_MIXER_B4: EQUIP_TYPE_8;
	EQUIP_TYPE_3_Valve2_RB4: EQUIP_TYPE_9;
	EQUIP_TYPE_3_Valve3_RB4: EQUIP_TYPE_9;
	EQUIP_TYPE_3_Valve4_RB4: EQUIP_TYPE_9;
	EQUIP_TYPE_9_Valve5_RB4: EQUIP_TYPE_9;
	EQUIP_TYPE_10_Dec_RB4: EQUIP_TYPE_10;
	reset_dec_RB4: BOOL;

	EQUP_TYPE_1_Pump_RB: EQUP_TYPE_1;
	reset_Pump2_RB: BOOL;

	sbr_airblower_A: EQUIPMENT_SBR_AIRBLOWER;
	sbr_airblower_B: EQUIPMENT_SBR_AIRBLOWER;

	(* sludge holding *)

	sludge_holding_A :sludge_holding;
	reset_polymer: BOOL;

	(*tertiary treatment *)
	tertiary_treatment_plant_A: tertiary_treatment_plant;

	(*reuse water*)
	REUSE_WATER_A: REUSE_WATER;




END_VAR
(*inlet*)
inlet();

(*sbr reactor*)
reactorA;
reactorB;


(*CHEMICAL*)
Chemical_A(
	iA1:= LSD210A_LimeTank1,
	iA2:= LSL210A_LimeTank1 ,
	iA3:= LSH210A_LimeTank1,
	iA4:= LSHH210A_LimeTank1,
	rA1:= reset_lime_tank_1,
	iB1:=LSD210B_LimeTank2 ,
	iB2:=LSL210B_LimeTank2 ,
	iB3:=LSH210B_LimeTank2 ,
	iB4:=LSHH210B_LimeTank2 ,
	rB1:=reset_lime_tank_2 ,
	iC1:= LSD210C_LimeTank3,
	iC2:= LSL210C_LimeTank3,
	iC3:= LSH210C_LimeTank3,
	iC4:= LSHH210C_LimeTank3,
	rC1:= reset_lime_tank_3,
	iqA2:= XV251A_LimeSelectorTank_OpenStat,
	iqB2:= XV251B_LimeSelectorTank_OpenStat,
	iqC2:= XV251C_LimeSelectorTank_OpenStat,
	iLRA:=XV221A_LimeValveR1_OpenStat OR XV222A_LimeValveR2_OpenStat OR XV223A_LimeValveR3_OpenStat OR XV224A_LimeValveR4_OpenStat ,
	iLRB:= XV221B_LimeValveR1_OpenStat OR XV222B_LimeValveR2_OpenStat OR XV223B_LimeValveR3_OpenStat OR XV224B_LimeValveR4_OpenStat  ,
	iAop1:= OPAlumA_AlumSelectorTank,
	iAop2:= OPAlumB_AlumSelectorTank,
	iAop3:= OPAlumC_AlumSelectorTank,
	iAop4:= OPAlumD_AlumSelectorTank,
	iAlss1:= LSL351A_AlumTank1,
	iAlss2:= LSL351B_AlumTank2 ,
	iAlss3:=LSL351C_AlumTank3 ,
	iAlss4:=LSL351D_AlumTank4 ,
	iasbrA:=XV211A_AlumValveR1_OpenStat OR XV212A_AlumValveR2_OpenStat OR XV213A_AlumValveR3_OpenStat OR XV214A_AlumValveR4_OpenStat,
	iasbrB:=XV211B_AlumValveR1_OpenStat OR XV212B_AlumValveR2_OpenStat OR XV213B_AlumValveR3_OpenStat OR XV214B_AlumValveR4_OpenStat,
	iCop1:= OPCausticA_CausticSodaSelectorTank1,
	iCop2:= OPCausticB_CausticSodaSelectorTank2,
	ilssC1:= LSL353A_CausticSodaTank,
	ilssC2:= LSL353B_CausticSodaTank,
	itpm:= P301A_EffluentTransferPump_RunStat,
	itpC:= ,
	itpCh:= ,
	ilssch1:=LSL355A_SodiumHypochloriteTank ,
	ilssch2:=LSL355A_SodiumHypochloriteTank ,
	ilssch3:=LSL355A_SodiumHypochloriteTank ,
	iChop1:= OPSodiumA_SodiumHypochloriteSelectorTank1,
	iChop2:= OPSodiumB_SodiumHypochloriteSelectorTank2,
	iChop3:= OPSodiumC_SodiumHypochloriteSelectorTank3,
	irdAB:= reactorA1.req_decanting OR reactorA2.req_decanting OR reactorA3.req_decanting OR reactorA4.req_decanting OR reactorB1.req_decanting OR reactorB2.req_decanting OR reactorB3.req_decanting OR reactorB4.req_decanting,
	qA1=> ,
	qA2=> ,
	qA3=> ,
	eA1=> ,
	qB1=> ,
	qB2=> ,
	qB3=> , 
	eB1=> , 
	qC1=> , 
	qC2=> , 
	qC3=> , 
	eC1=> , 
	qD1=> , 
	qD2=> , 
	qD3=> , 
	eD1=> , 
	qCir=> ,
	qLA=> , 
	qLB=> , 
	qP1=> , 
	qP2=> , 
	qP3=> , 
	qP4=> ,
	qtA1=> , 
	qtC1=> , 
	qtCH1=> , 
	qdsp=> );

(*sludge holding*)
sludge_holding_A(
	i1A:= LSL501A_SludgeStorage,
	i1B:= LSL501B_SludgeStorage,
	i2A:= LSH501A_SludgeStorage,
	i2B:= LSH501B_SludgeStorage,
	i3A:=LSHH501A_SludgeStorage ,
	i3B:=LSHH501B_SludgeStorage,
	i4:= LSL309A_WaterLevelTank ,
	i5:= LSHPU501_PolymerTankLevel,
	i6:= LSLPU501_PolymerTankLevel,
	i7:= LSH600_SludgePitSensor > 30,
	ic1:=(*blower*) ,
	ic2:= ,
	s1:=(*to complete with drum and backwash*)  ,
	s2:=M503_PolymerStirrer_EStopStat OR M503_PolymerStirrer_OverloadStat ,
	s3:= ,
	s4:= B501A_Blower_IncompleteStat OR B501A_Blower_OverloadStat OR B501A_Blower_EStopStat,
	s5:=  B501B_Blower_IncompleteStat OR B501B_Blower_OverloadStat OR B501B_Blower_EStopStat ,
	r1:= reset_polymer,
	q1A=> , 
	q2A=> , 
	q1B=> ,
	q2B=> , 
	q3=> , 
	q4=> , 
	q5=> ,
	q6=> , 
	q7=> , 
	q8=> , 
	q9=> , 
	q10=> , 
	q11=> , 
	q12=> , 
	q13=> , 
	q14=> , 
	c1=> , 
	e1=> );

(*tertiary treatment*)
tertiary_treatment_plant_A(
	i1:= LSH301_EffluentSump,
	i2:= LSL309A_WaterLevelTank,
	i3:= LSL301_EffluentSump,
	i4:= (*not applicable*),
	i5:= LSH302_CollectionSump,
	i6:= LSH501A_SludgeStorage AND LSH501B_SludgeStorage,
	i7:= LSHH501A_SludgeStorage AND LSHH501B_SludgeStorage,
	s1:= K301A_AirCompressor_RunStat,
	s2:= K301B_AirCompressor_RunStat,
	s3:= P301A_EffluentTransferPump_RunStat,
	s4:= P301B_EffluentTransferPump_RunStat ,
	q1=> , 
	q2=> , 
	q3=> , 
	q4=> , 
	q5=> , 
	q6=> , 
	q7=> , 
	q8=> ,
	q9=> , 
	q10=> , 
	q11=> , 
	q12=> );

(*reuse water*)
REUSE_WATER_A(
	i3:= PSL412_PressureSwitch,
	i1:= LSL309A_WaterLevelTank,
	i4:= LSH405_VacuumChestLevel,
	i2:= (*unused*),
	i5:= PG413_LowPressureGauge,
	i6:= PG414_HighPressureGauge,
	p1:= PSL411_PressureTransmitter,
	q1=> ,
	q2=> ,
	q3=> , 
	q4=> , 
	q5=> , 
	q6=> , 
	q7=> , 
	q8=> , 
	q9=> );



(*0-60 bar fra 4-20 mA resolution 0.1 bar:

FACTOR = 10
Data @ 4 mA = 6240
Data @ 20 mA = 31208
DataOffset = 6240
DataSpan = 31208 - 6240 = 24968
EUOffset = 0 x 10 = 0
EUSpan = (60 - 0) x 10 = 600

DATA = 18975

EU = ((600 x (18975 - 6240)) / 24968) + 0 = 306

Process value = 306 / 10 = 30.6 bar *)
AT300_EffluentTurbidityEntry_ScaledValue:=REAL_TO_INT(AT300_EffluentTurbidityEntry);
AT302_TreatedEffluentTurbidityDischarge_ScaledValue:=REAL_TO_INT(AT302_TreatedEffluentTurbidityDischarge);
CL303_ResidualChlorineAnalyzer_ScaledValue:=REAL_TO_INT(CL303_ResidualChlorineAnalyzer);
CL304_FinalChlorineAnalyzer_ScaledValue:=REAL_TO_INT(CL304_FinalChlorineAnalyzer);
D0201A4_DOProfilesR4_ScaledValue:=REAL_TO_INT(D0201A4_DOProfilesR4);
D0201B4_DOProfilesR4_ScaledValue:=REAL_TO_INT(D0201B4_DOProfilesR4);
DO201A1_DOProfilesR1_ScaledValue:=REAL_TO_INT(DO201A1_DOProfilesR1);
DO201A2_DOProfilesR2_ScaledValue:=REAL_TO_INT(DO201A2_DOProfilesR2);
DO201A3_DOProfilesR3_ScaledValue:=REAL_TO_INT(DO201A3_DOProfilesR3);
DO201B1_DOProfilesR1_ScaledValue:=REAL_TO_INT(DO201B1_DOProfilesR1);
DO201B2_DOProfilesR2_ScaledValue:=REAL_TO_INT(DO201B2_DOProfilesR2);
DO201B3_DOProfilesR3_ScaledValue:=REAL_TO_INT(DO201B3_DOProfilesR3);
FT100A_FlowTotalizerS1_ScaledValue:=REAL_TO_INT(FT100A_FlowTotalizerS1);
FT100B_FlowTotalizerS2_ScaledValue:=REAL_TO_INT(FT100B_FlowTotalizerS2);
FT300_EffluentFlowrateEntry_ScaledValue:=REAL_TO_INT(FT300_EffluentFlowrateEntry);
FT301_TreatedEffluentFlowrateDischarge_ScaledValue:=REAL_TO_INT(FT301_TreatedEffluentFlowrateDischarge);
LSH600_SludgePitSensor_ScaledValue:=REAL_TO_INT(LSH600_SludgePitSensor);
ORP_DisinfectionTankAnalyzer_ScaledValue:=REAL_TO_INT(ORP_DisinfectionTankAnalyzer);
PHT201A1_pHlevelR1_ScaledValue:=REAL_TO_INT(PHT201A1_pHlevelR1);
PHT201A2_pHlevelR2_ScaledValue:=REAL_TO_INT(PHT201A2_pHlevelR2);
PHT201A3_pHlevelR3_ScaledValue:=REAL_TO_INT(PHT201A3_pHlevelR3);
PHT201A4_pHlevelR4_ScaledValue:=REAL_TO_INT(PHT201A4_pHlevelR4);
PHT201B1_pHlevelR1_ScaledValue:=REAL_TO_INT(PHT201B1_pHlevelR1);
PHT201B2_pHlevelR2_ScaledValue:=REAL_TO_INT(PHT201B2_pHlevelR2);
PHT201B3_pHlevelR3_ScaledValue:=REAL_TO_INT(PHT201B3_pHlevelR3);
PHT201B4_pHlevelR4_ScaledValue:=REAL_TO_INT(PHT201B4_pHlevelR4);
PHT301_EffluentpHLevelEntry_ScaledValue:=REAL_TO_INT(PHT301_EffluentpHLevelEntry);
PHT303_TreatedEffluentpHLevelDischarge_ScaledValue:=REAL_TO_INT(PHT303_TreatedEffluentpHLevelDischarge);
PSL411_PressureTransmitter_ScaledValue:=REAL_TO_INT(PSL411_PressureTransmitter);

AUX902_PLCRunStatus:=TRUE;
IF GENRUN_Generator_RunStat=TRUE THEN
	AUX903_GeneratorSupplyStat:=TRUE;
ELSE
	AUX903_GeneratorSupplyStat:=FALSE;
END_IF

IF GENFAIL_Generator_FailStat=TRUE OR GENOT_Generator_OverloadStat=TRUE THEN
	AUX901_CommonAlarm:=TRUE;
END_IF

IF GENFAIL_Generator_FailStat=FALSE AND GENOT_Generator_OverloadStat=FALSE THEN
	AUX901_CommonAlarm:=FALSE;
END_IF

IF ScadaRoom_KouplerUTP_State=8 THEN
	ScadaRoom_KouplerUTP_StateBool:=TRUE;
ELSE
	ScadaRoom_KouplerUTP_StateBool:=FALSE;
END_IF

IF ScadaRoom_KouplerFiber_State=8 THEN
	ScadaRoom_KouplerFiber_StateBool:=TRUE;
ELSE
	ScadaRoom_KouplerFiber_StateBool:=FALSE;
END_IF

IF InletWork_1_KouplerFiber_State=8 THEN
	InletWork_1_KouplerFiber_StateBool:=TRUE;
ELSE
	InletWork_1_KouplerFiber_StateBool:=FALSE;
END_IF

IF InletWork_2_KouplerFiber_State=8 THEN
	InletWork_2_KouplerFiber_StateBool:=TRUE;
ELSE
	InletWork_2_KouplerFiber_StateBool:=FALSE;
END_IF

IF BlowerHouse_2_KouplerFiber_State=8 THEN
	BlowerHouse_2_KouplerFiber_StateBool:=TRUE;
ELSE
	BlowerHouse_2_KouplerFiber_StateBool:=FALSE;
END_IF

IF BlowerHouse_1_KouplerFiber_State=8 THEN
	BlowerHouse_1_KouplerFiber_StateBool:=TRUE;
ELSE
	BlowerHouse_1_KouplerFiber_StateBool:=FALSE;
END_IF

IF SBR_1_KouplerFiber_State=8 THEN
	SBR_1_KouplerFiber_StateBool:=TRUE;
ELSE
	SBR_1_KouplerFiber_StateBool:=FALSE;
END_IF

IF SBR_2_KouplerFiber_State=8 THEN
	SBR_2_KouplerFiber_StateBool:=TRUE;
ELSE
	SBR_2_KouplerFiber_StateBool:=FALSE;
END_IF

IF ChemicalAndTertiary_KouplerFiber_State=8 THEN
	ChemicalAndTertiary_KouplerFiber_StateBool:=TRUE;
ELSE
	ChemicalAndTertiary_KouplerFiber_StateBool:=FALSE;
END_IF

IF SludgeThickening_KouplerFiber_State=8 THEN
	SludgeThickening_KouplerFiber_StateBool:=TRUE;
ELSE
	SludgeThickening_KouplerFiber_StateBool:=FALSE;
END_IF

IF Reused_KouplerFiber_State=8 THEN
	Reused_KouplerFiber_StateBool:=TRUE;
ELSE
	Reused_KouplerFiber_StateBool:=FALSE;
END_IF

IF ScadaRoom_KouplerFiber_Return_State=8 THEN
	ScadaRoom_KouplerFiber_Return_StateBool:=TRUE;
ELSE
	ScadaRoom_KouplerFiber_Return_StateBool:=FALSE;
END_IF
END_PROGRAM
ACTION inlet:
(*INLET A*)
INLET_A(
	i1:= LSL101A_EQFloatSensor,
	i3:= LSHH103A_SBRFloatSensor,
	i2:= LSH101A_EQFloatSensor,
	i4:= LSHH105A2_StreamLineOverflow,
	i5:= LSL100A_MixerFloatSensor,
	i6:= LSH100A_MixerFloatSensor,
	r1:= rA1,
	i7:= PS101A1_Penstock_OpenStat,
	i8:= PS101A2_Penstock_OpenStat,
	i10:= LSHH105A2_StreamLineOverflow,
	i11:= LSH105A1_StreamLineFlow,
	s1:= F101A1_FineScr_EStopStat,
	s2:= F101A1_FineScr_OverloadStat,
	s3:=F101A2_FineScr_EStopStat ,
	s4:=F101A2_FineScr_OverloadStat ,
	i12:=LSL103A_SBRFloatSensor ,
	i13:=LSH103A_SBRFloatSensor );

EQUIP_TYPE_1_EQA(
	i1:=INLET_A.q1 ,
	i2:= INLET_A.q2,
	r1:= r_eqA1,
	sa1:= P101A1_EQPump_EStopStat ,
	sa2:= P101A1_EQPump_IncompleteStat ,
	sa3:= P101A1_EQPump_LocalRemoteStat ,
	sa4:= P101A1_EQPump_OverloadStat ,
	sa5:= P101A1_EQPump_RunStat,
	sb1:= P101A2_EQPump_EStopStat ,
	sb2:= P101A2_EQPump_IncompleteStat ,
	sb3:= P101A2_EQPump_LocalRemoteStat,
	sb4:= P101A2_EQPump_OverloadStat  ,
	sb5:= P101A2_EQPump_RunStat,
	c1=> ,
	c2=> ,
	q1=>P101A1_EQPump_RunCmd ,
	q2=>P101A2_EQPump_RunCmd ,
	e1=> );

EQUIP_TYPE_2_MXA(
	i1:= INLET_A.q3,
	i2:= INLET_A.q4,
	sa1:= M101A1_EQMixer_EStopStat,
	sa2:= M101A1_EQMixer_IncompleteStat,
	sa3:= M101A1_EQMixer_LocalRemoteStat,
	sa4:= M101A1_EQMixer_OverloadStat,
	sa5:= M101A1_EQMixer_RunStat,
	sb1:= M101A2_EQMixer_EStopStat,
	sb2:= M101A2_EQMixer_IncompleteStat,
	sb3:= M101A2_EQMixer_LocalRemoteStat,
	sb4:= M101A2_EQMixer_OverloadStat,
	sb5:= M101A2_EQMixer_RunStat,
	c1=> ,
	q1=> M101A1_EQMixer_RunCmd,
	q2=> M101A2_EQMixer_RunCmd,
	e1=> );

EQUIP_TYPE_3_PSA1(
	i1:= NOT INLET_A.q5,
	i2:= INLET_A.q5,
	s1:=PS101A1_Penstock_CloseStat ,
	s2:= PS101A1_Penstock_LocalRemoteStat,
	s3:=PS101A1_Penstock_OpenStat ,
	s4:=PS101A1_Penstock_TripStat ,
	c1=> ,
	q1=>PS101A1_Penstock_CloseCmd ,
	q2=>PS101A1_Penstock_OpenCmd );


EQUIP_TYPE_3_PSA2(
	i1:= NOT INLET_A.q6,
	i2:= INLET_A.q6,
	s1:=PS101A2_Penstock_CloseStat ,
	s2:= PS101A2_Penstock_LocalRemoteStat,
	s3:=PS101A2_Penstock_OpenStat ,
	s4:=PS101A2_Penstock_TripStat ,
	c1=> ,
	q1=>PS101A2_Penstock_CloseCmd ,
	q2=>PS101A2_Penstock_OpenCmd );

EQUIP_TYPE_4_SPA(
	i1:= INLET_A.q9,
	i2:=INLET_A.q10 ,
	sa1:=C101A_ScreenCompactor_EStopStat ,
	sa2:= C101A_ScreenCompactor_LocalRemoteStat,
	sa3:= C101A_ScreeningCompactor_OverloadStat,
	sa4:= C101A_ScreenCompactor_RunStat,
	c1=> ,
	q1=> C101A_ScreenCompactor_RunCmd,
	e1=> );

EQUIP_TYPE_4_SCA(
	i1:=INLET_A.q7,
	i2:= INLET_A.q8,
	sa1:= C102A_ScreenConveyer_EStopStat,
	sa2:= C102A_ScreenConveyer_LocalRemoteStat,
	sa3:= C102A_ScreeningConveyer_OverloadStat,
	sa4:= C102A_ScreenConveyer_RunStat,
	c1=> ,
	q1=> C102A_ScreenConveyer_RunCmd,
	e1=> );

EQUIP_TYPE_5_CWSA(
	i1:=INLET_A.q11 ,
	i2:=INLET_A.q12 ,
	sa1:= XV102A1_ContinuosValveWater_CloseStat,
	sa2:=XV102A1_ContinuosValveWater_OpenStat ,
	c1=> ,
	q1=> XV102A1_ContinuosValveWater_OpenCmd,
	e1=> );

EQUIP_TYPE_4_FSA1(
	i1:= INLET_A.q13,
	i2:= INLET_A.q14,
	sa1:= F101A1_FineScr_EStopStat,
	sa2:= F101A1_FineScr_LocalRemoteStat,
	sa3:= F101A1_FineScr_OverloadStat,
	sa4:= F101A1_FineScr_RunStat,
	c1=> ,
	q1=> F101A1_FineScr_RunCmd,
	e1=> );


EQUIP_TYPE_4_FSA2(
	i1:= INLET_A.q15,
	i2:= INLET_A.q16,
	sa1:= F101A2_FineScr_EStopStat,
	sa2:= F101A2_FineScr_LocalRemoteStat,
	sa3:= F101A2_FineScr_OverloadStat,
	sa4:= F101A2_FineScr_RunStat,
	c1=> ,
	q1=> F101A2_FineScr_RunCmd,
	e1=> );


EQUIP_TYPE_6_WSA1(
	i1:=INLET_A.q17 ,
	i2:=INLET_A.q18 ,
	sa1:=XV101A1_SolenoidValveSpray_CloseStat ,
	sa2:=XV101A1_SolenoidValveSpray_OpenStat ,
	c1=> ,
	q1=>XV101A1_SolenoidValveSpray_OpenCmd ,
	e1=> );

EQUIP_TYPE_6_WSA2(
	i1:=INLET_A.q19 ,
	i2:=INLET_A.q20 ,
	sa1:=XV101A2_SolenoidValveSpray_CloseStat ,
	sa2:=XV101A2_SolenoidValveSpray_OpenStat ,
	c1=> ,
	q1=>XV101A2_SolenoidValveSpray_OpenCmd ,
	e1=> );

EQUIP_TYPE_5_GRVA1(
	i1:=NOT INLET_A.q21 ,
	i2:=INLET_A.q21 ,
	sa1:=XV100A1_GritRemovalValve_CloseStat ,
	sa2:=XV100A1_GritRemovalValve_OpenStat ,
	c1=> XV100A1_GritRemovalValve_OpenCmd,
	q1=> ,
	e1=> );


EQUIP_TYPE_5_GRVA2(
	i1:=NOT INLET_A.q22 ,
	i2:=INLET_A.q22 ,
	sa1:=XV100A2_GritRemovalValve_CloseStat ,
	sa2:=XV100A2_GritRemovalValve_OpenStat ,
	c1=> XV100A1_GritRemovalValve_OpenCmd,
	q1=> ,
	e1=> );


EQUIP_TYPE_4_ClassifierA(
	i1:=INLET_A.q25 ,
	i2:=INLET_A.q26 ,
	sa1:=C103A_GritClasifier_EStopStat ,
	sa2:= C103A_GritClasifier_LocalRemoteStat,
	sa3:= C103A_GritClasifier_RunStat,
	sa4:= C103A_GritClassifier_OverloadStat,
	c1=> ,
	q1=>C103A_GritClasifier_RunCmd ,
	e1=> );

EQUP_TYPE_1_STA1(
	i1:=INLET_A.q27 ,
	i2:=INLET_A.q28 ,
	r1:=r_STA1 ,
	sa1:=P102A1_SBRTransferPump_EStopStat ,
	sa2:=P102A1_SBRTransferPump_IncompleteStat ,
	sa3:=P102A1_SBRTransferPump_LocalRemoteStat ,
	sa4:=P102A1_SBRTransferPump_OverloadStat ,
	sa5:=P102A1_SBRTransferPump_RunStat ,
	sb1:=P102A2_SBRTransferPump_EStopStat ,
	sb2:=P102A2_SBRTransferPump_IncompleteStat ,
	sb3:=P102A2_SBRTransferPump_LocalRemoteStat ,
	sb4:=P102A2_SBRTransferPump_OverloadStat ,
	sb5:=P102A2_SBRTransferPump_RunStat ,
	c1=> ,
	c2=> ,
	q1=>P102A1_SBRTransferPump_RunCmd ,
	q2=>P102A2_SBRTransferPump_RunCmd ,
	e1=> );

(* INLET B *)
INLET_B(
	i1:= LSL101B_EQFloatSensor,
	i3:= LSHH103B_SBRFloatSensor,
	i2:= LSH101B_EQFloatSensor,
	i4:= LSHH105B2_StreamLineOverflow,
	i5:= LSL100B_MixerFloatSensor,
	i6:= LSH100B_MixerFloatSensor,
	r1:= rB1,
	i7:= PS101B1_Penstock_OpenStat,
	i8:= PS101B2_Penstock_OpenStat,
	i10:= LSHH105B2_StreamLineOverflow,
	i11:= LSH105B1_StreamLineFlow,
	s1:= F101B1_FineScr_EStopStat,
	s2:= F101B1_FineScr_OverloadStat,
	s3:=F101B2_FineScr_EStopStat ,
	s4:=F101B2_FineScr_OverloadStat ,
	i12:=LSL103B_SBRFloatSensor ,
	i13:=LSH103B_SBRFloatSensor );

EQUIP_TYPE_1_EQB(
	i1:=INLET_B.q1 ,
	i2:= INLET_B.q2,
	r1:= r_eqB1,
	sa1:= P101B1_EQPump_EStopStat ,
	sa2:= P101B1_EQPump_IncompleteStat ,
	sa3:= P101B1_EQPump_LocalRemoteStat ,
	sa4:= P101B1_EQPump_OverloadStat ,
	sa5:= P101B1_EQPump_RunStat,
	sb1:= P101B2_EQPump_EStopStat ,
	sb2:= P101B2_EQPump_IncompleteStat ,
	sb3:= P101B2_EQPump_LocalRemoteStat,
	sb4:= P101B2_EQPump_OverloadStat  ,
	sb5:= P101B2_EQPump_RunStat,
	c1=> ,
	c2=> ,
	q1=>P101B1_EQPump_RunCmd ,
	q2=>P101B2_EQPump_RunCmd ,
	e1=> );

EQUIP_TYPE_2_MXB(
	i1:= INLET_B.q3,
	i2:= INLET_B.q4,
	sa1:= M101B1_EQMixer_EStopStat,
	sa2:= M101B1_EQMixer_IncompleteStat,
	sa3:= M101B1_EQMixer_LocalRemoteStat,
	sa4:= M101B1_EQMixer_OverloadStat,
	sa5:= M101B1_EQMixer_RunStat,
	sb1:= M101B2_EQMixer_EStopStat,
	sb2:= M101B2_EQMixer_IncompleteStat,
	sb3:= M101B2_EQMixer_LocalRemoteStat,
	sb4:= M101B2_EQMixer_OverloadStat,
	sb5:= M101B2_EQMixer_RunStat,
	c1=> ,
	q1=> M101B1_EQMixer_RunCmd,
	q2=> M101B2_EQMixer_RunCmd,
	e1=> );

EQUIP_TYPE_3_PSB1(
	i1:= NOT INLET_B.q5,
	i2:= INLET_B.q5,
	s1:=PS101B1_Penstock_CloseStat ,
	s2:= PS101B1_Penstock_LocalRemoteStat,
	s3:=PS101B1_Penstock_OpenStat ,
	s4:=PS101B1_Penstock_TripStat ,
	c1=> ,
	q1=>PS101B1_Penstock_CloseCmd ,
	q2=>PS101B1_Penstock_OpenCmd );


EQUIP_TYPE_3_PSB2(
	i1:= NOT INLET_B.q6,
	i2:= INLET_B.q6,
	s1:=PS101B2_Penstock_CloseStat ,
	s2:= PS101B2_Penstock_LocalRemoteStat,
	s3:=PS101B2_Penstock_OpenStat ,
	s4:=PSB101B2_Penstock_TripStat,
	c1=> ,
	q1=>PS101B2_Penstock_CloseCmd ,
	q2=>PS101B2_Penstock_OpenCmd );

EQUIP_TYPE_4_SPB(
	i1:= INLET_B.q9,
	i2:=INLET_B.q10 ,
	sa1:=C101B_ScreenCompactor_EStopStat ,
	sa2:= C101B_ScreenCompactor_LocalRemoteStat,
	sa3:= C101B_ScreeningCompactor_OverloadStat,
	sa4:= C101B_ScreenCompactor_RunStat,
	c1=> ,
	q1=> C101B_ScreenCompactor_RunCmd,
	e1=> );

EQUIP_TYPE_4_SCB(
	i1:=INLET_B.q7,
	i2:= INLET_B.q8,
	sa1:= C102B_ScreenConveyer_EStopStat,
	sa2:= C102B_ScreenConveyer_LocalRemoteStat,
	sa3:= C102B_ScreeningConveyer_OverloadStat,
	sa4:= C102B_ScreenConveyer_RunStat,
	c1=> ,
	q1=> C102B_ScreenConveyer_RunCmd,
	e1=> );

EQUIP_TYPE_5_CWSB(
	i1:=INLET_B.q11 ,
	i2:=INLET_B.q12 ,
	sa1:= XV102B1_ContinuosValveWater_CloseStat,
	sa2:=XV102B1_ContinuosValveWater_OpenStat ,
	c1=> ,
	q1=> XV102B1_ContinuosValveWater_OpenCmd,
	e1=> );

EQUIP_TYPE_4_FSB1(
	i1:= INLET_B.q13,
	i2:= INLET_B.q14,
	sa1:= F101B1_FineScr_EStopStat,
	sa2:= F101B1_FineScr_LocalRemoteStat,
	sa3:= F101B1_FineScr_OverloadStat,
	sa4:= F101B1_FineScr_RunStat,
	c1=> ,
	q1=> F101B1_FineScr_RunCmd,
	e1=> );


EQUIP_TYPE_4_FSB2(
	i1:= INLET_B.q15,
	i2:= INLET_B.q16,
	sa1:= F101B2_FineScr_EStopStat,
	sa2:= F101B2_FineScr_LocalRemoteStat,
	sa3:= F101B2_FineScr_OverloadStat,
	sa4:= F101B2_FineScr_RunStat,
	c1=> ,
	q1=> F101B2_FineScr_RunCmd,
	e1=> );


EQUIP_TYPE_6_WSB1(
	i1:=INLET_B.q17 ,
	i2:=INLET_B.q18 ,
	sa1:=XV101B1_SolenoidValveSpray_CloseStat ,
	sa2:=XV101B1_SolenoidValveSpray_OpenStat ,
	c1=> ,
	q1=>XV101B1_SolenoidValveSpray_OpenCmd ,
	e1=> );

EQUIP_TYPE_6_WSB2(
	i1:=INLET_B.q19 ,
	i2:=INLET_B.q20 ,
	sa1:=XV101B2_SolenoidValveSpray_CloseStat ,
	sa2:=XV101B2_SolenoidValveSpray_OpenStat ,
	c1=> ,
	q1=>XV101B2_SolenoidValveSpray_OpenCmd ,
	e1=> );

EQUIP_TYPE_5_GRVB1(
	i1:=NOT INLET_B.q21 ,
	i2:=INLET_B.q21 ,
	sa1:=XV100B1_GritRemovalValve_CloseStat ,
	sa2:=XV100B1_GritRemovalValve_OpenStat ,
	c1=> XV100B1_GritRemovalValve_OpenCmd,
	q1=> ,
	e1=> );


EQUIP_TYPE_5_GRVB2(
	i1:=NOT INLET_B.q22 ,
	i2:=INLET_B.q22 ,
	sa1:=XV100B2_GritRemovalValve_CloseStat ,
	sa2:=XV100B2_GritRemovalValve_OpenStat ,
	c1=> XV100B1_GritRemovalValve_OpenCmd,
	q1=> ,
	e1=> );


EQUIP_TYPE_4_ClassifierB(
	i1:=INLET_B.q25 ,
	i2:=INLET_B.q26 ,
	sa1:=C103B_GritClasifier_EStopStat ,
	sa2:= C103BB_GritClasifiier_LocalRemoteStat,
	sa3:= C103B_GritClasifier_RunStat,
	sa4:= C103B_GritClassifier_OverloadStat,
	c1=> ,
	q1=>C103B_GritClasifier_RunCmd ,
	e1=> );

EQUP_TYPE_1_STB1(
	i1:=INLET_B.q27 ,
	i2:=INLET_B.q28 ,
	r1:=r_STB1 ,
	sa1:=P102B1_SBRTransferPump_EStopStat ,
	sa2:=P102B1_SBRTransferPump_IncompleteStat ,
	sa3:=P102B1_SBRTransferPump_LocalRemoteStat ,
	sa4:=P102B1_SBRTransferPump_OverloadStat ,
	sa5:=P102B1_SBRTransferPump_RunStat ,
	sb1:=P102B2_SBRTransferPump_EStopStat ,
	sb2:=P102B2_SBRTransferPump_IncompleteStat ,
	sb3:=P102B2_SBRTransferPump_LocalRemoteStat ,
	sb4:=P102B2_SBRTransferPump_OverloadStat ,
	sb5:=P102B2_SBRTransferPump_RunStat ,
	c1=> ,
	c2=> ,
	q1=>P102B1_SBRTransferPump_RunCmd ,
	q2=>P102B2_SBRTransferPump_RunCmd ,
	e1=> );

(*EQ blower*)
EQUP_TYPE_7_Blower(
	i1:=INLET_A.q23 AND INLET_B.q23,
	i2:= INLET_A.q24 OR INLET_B.q24,
	r1:=rblower ,
	sa1:= B101A1_AirBlower_EStopStat,
	sa2:= B101A1_AirBlower_IncompleteStat ,
	sa3:= B101A1_AirBlower_LocalRemoteStat,
	sa4:= B101A1_AirBlower_OverloadStat ,
	sa5:= B101A1_AirBlower_OnOffStat,
	sb1:= B101A2_AirBlower_EStopStat,
	sb2:= B101A2_AirBlower_IncompleteStat ,
	sb3:= B101A2_AirBlower_LocalRemoteStat,
	sb4:= B101A2_AirBlower_OverloadStat ,
	sb5:= B101A2_AirBlower_OnOffStat,
	c1=> ,
	c2=> ,
	q1=> B101A1_AirBlower_RunCmd,
	q2=> B101A2_AirBlower_RunCmd,
	e1=> );
END_ACTION
ACTION reactorA:
(*REACTOR A*)

reactorA1(
	op:= OPR1A_ReactorStatus,
	res_fill:=Fill_selectorA.q1 ,
	i1:= LSH201A1_LevelSensorR1 ,
	alum_time:= Alum_reactorA1,
	res_aeration:= Aerate_selectorA.q1,
	ph1:=PHT201A1_pHlevelR1 ,
	res_decanting:=Decant_selectorA.q1 ,
	r1:=resumeAlumA1 ,
	i2:=LSHH501A_SludgeStorage ,
	i3:=HR201A1_DecantHighLevelR1 ,
	i4:=LR201A1_DecantLowLevelR1 ,
	req_fill=> ,
	q1=> ,
	q2=> ,
	q4=> ,
	q3=> ,
	q5=> ,
	q6=> ,
	req_aeration=> ,
	e1=> ,
	q7=> ,
	q8=> ,
	m1=> ,
	req_settle=> ,
	req_decanting=> ,
	q9=> );

reactorA2(
	op:= OPR2A_ReactorStatus,
	res_fill:=Fill_selectorA.q2 ,
	i1:= LSH201A2_LevelSensorR2 ,
	alum_time:= Alum_reactorA2,
	res_aeration:= Aerate_selectorA.q2,
	ph1:=PHT201A2_pHlevelR2 ,
	res_decanting:=Decant_selectorA.q2 ,
	r1:=resumeAlumA2 ,
	i2:=LSHH501A_SludgeStorage ,
	i3:=HR201A2_DecantHighLevelR2 ,
	i4:=LR201A2_DecantLowLevelR2 ,
	req_fill=> ,
	q1=> ,
	q2=> ,
	q4=> ,
	q3=> ,
	q5=> ,
	q6=> ,
	req_aeration=> ,
	e1=> ,
	q7=> ,
	q8=> ,
	m1=> ,
	req_settle=> ,
	req_decanting=> ,
	q9=> );

reactorA3(
	op:= OPR3A_ReactorStatus,
	res_fill:=Fill_selectorA.q3 ,
	i1:= LSH201A3_LevelSensorR3 ,
	alum_time:= Alum_reactorA3,
	res_aeration:= Aerate_selectorA.q3,
	ph1:=PHT201A3_pHlevelR3 ,
	res_decanting:=Decant_selectorA.q3 ,
	r1:=resumeAlumA3 ,
	i2:=LSHH501A_SludgeStorage ,
	i3:=HR201A3_DecantHighLevelR3 ,
	i4:=LR201A3_DecantLowLevelR3 ,
	req_fill=> ,
	q1=> ,
	q2=> ,
	q4=> ,
	q3=> ,
	q5=> ,
	q6=> ,
	req_aeration=> ,
	e1=> ,
	q7=> ,
	q8=> ,
	m1=> ,
	req_settle=> ,
	req_decanting=> ,
	q9=> );

reactorA4(
	op:= OPR4A_ReactorStatus,
	res_fill:=Fill_selectorA.q4 ,
	i1:= LSH201A4_LevelSensorR4 ,
	alum_time:= Alum_reactorA4,
	res_aeration:= Aerate_selectorA.q4,
	ph1:=PHT201A4_pHlevelR4 ,
	res_decanting:=Decant_selectorA.q4 ,
	r1:=resumeAlumA4 ,
	i2:=LSHH501A_SludgeStorage ,
	i3:=HR201A4_DecantHighLevelR4 ,
	i4:=LR201A4_DecantLowLevelR4 ,
	req_fill=> ,
	q1=> ,
	q2=> ,
	q4=> ,
	q3=> ,
	q5=> ,
	q6=> ,
	req_aeration=> ,
	e1=> ,
	q7=> ,
	q8=> ,
	m1=> ,
	req_settle=> ,
	req_decanting=> ,
	q9=> );

fill_selectorA(
	i1:=ReactorA1.req_fill ,
	i2:=ReactorA2.req_fill ,
	i3:=ReactorA3.req_fill ,
	i4:=ReactorA4.req_fill,
	q1=> ,
	q2=> ,
	q3=> ,
	q4=> ,
	c1=> );

aerate_selectorA(
	i1:=ReactorA1.req_aeration,
	i2:=ReactorA2.req_aeration ,
	i3:=ReactorA3.req_aeration ,
	i4:=ReactorA4.req_aeration ,
	available:=2 ,
	q1=> ,
	q2=> ,
	q3=> ,
	q4=>);

decant_selectorA(
	i1:=  ReactorA1.req_decanting,
	i2:=  ReactorA2.req_decanting,
	i3:=  ReactorA3.req_decanting,
	i4:=  ReactorA4.req_decanting,
	q1=> ,
	q2=> ,
	q3=> ,
	q4=> ,
	c1=> );

sbr_airblower_A(
	sa1:= B201A1_AirBlowerS1_EStopStat,
	sa2:= B201A1_AirBlowerS1_IncompleteStat,
	sa3:= B201A1_AirBlowerS1_LocalRemoteStat,
	sa4:= B201A1_AirBlowerS1_OverloadStat,
	sa5:= B201A1_AirBlowerS1_RunStat,
	sb1:= B201A2_AirBlowerS1_EStopStat,
	sb2:= B201A2_AirBlowerS1_IncompleteStat,
	sb3:= B201A2_AirBlowerS1_LocalRemoteStat,
	sb4:= B201A2_AirBlowerS1_OverloadStat,
	sb5:= B201A2_AirBlowerS1_RunStat,
	sc1:= B201A3_AirBlowerS1_EStopStat,
	sc2:= B201A3_AirBlowerS1_IncompleteStat,
	sc3:= B201A3_AirBlowerS1_LocalRemoteStat,
	sc4:= B201A3_AirBlowerS1_OverloadStat,
	sc5:= B201A3_AirBlowerS1_RunStat,
	req:= aerate_selectorA.taken,
	q1=> B201A1_AirBlowerS1_RunCmd,
	q2=> B201A2_AirBlowerS1_RunCmd,
	q3=> B201A3_AirBlowerS1_RunCmd);


EQUP_TYPE_1_Pump_RA(
	i1:= NOT( reactorA1.q6 AND reactorA2.q6 AND reactorA3.q6 AND reactorA4.q6),
	i2:= reactorA1.q6 OR reactorA2.q6 OR reactorA3.q6 OR reactorA4.q6,
	r1:= reset_Pump2_RA,
	sa1:=P201A1_DesludgePumpS1_EStopStat ,
	sa2:= ,
	sa3:=P201A1_DesludgePumpS1_LocalRemoteStat ,
	sa4:= P201A1_DesludgePumpS1_OverloadStatus,
	sa5:=P201A1_DesludgePumpS1_RunStat ,
	sb1:= P201A2_DesludgePumpS1_EStopStat,
	sb2:= ,
	sb3:=P201A2_DesludgePumpS1_LocalRemoteStat ,
	sb4:= P201A2_DesludgePumpS1_OverloadStatus,
	sb5:=P201A2_DesludgePumpS1_RunStat ,
	c1=> ,
	c2=> ,
	q1=>P201A1_DesludgePump_RunCmd,
	q2=>P201A2_DesludgePump_RunCmd ,
	e1=> );


EQUIP_TYPE_3_Valva1_RA1(
	i1:=NOT reactorA1.q1 ,
	i2:=reactorA1.q1 ,
	s1:=XV205A_SBRValveR1_CloseStat ,
	s2:=XV205A_SBRValveR1_OpenStat ,
	c1=> ,
	q1=>XV205A_SBRValveR1_CloseCmd ,
	q2=>XV205A_SBRValveR1_OpenCmd);

EQUIP_TYPE_8_MIXER_A1(
	i1:= NOT reactorA1.q2,
	i2:= reactorA1.q2,
	sa1:=M200A1A_MixerR1_EStopStat,
	sa2:=M200A1A_MixerR1_IncompleteStat ,
	sa3:=M200A1A_MixerR1_LocalRemoteStat ,
	sa4:=M200A1A_MixerR1_OverloadStat ,
	sa5:=M200A1A_MixerR1_RunStat ,
	sb1:=M200A1B_MixerR1_EStopStat,
	sb2:=M200A1B_MixerR1_IncompleteStat ,
	sb3:=M200A1B_MixerR1_LocalRemoteStat ,
	sb4:=M200A1B_MixerR1_OverloadStat ,
	sb5:=M200A1B_MixerR1_RunStat ,
	sc1:=M200A1C_MixerR1_EStopStat,
	sc2:=M200A1C_MixerR1_IncompleteStat ,
	sc3:=M200A1C_MixerR1_LocalRemoteStat ,
	sc4:=M200A1C_MixerR1_OverloadStat ,
	sc5:=M200A1C_MixerR1_RunStat ,
	c1=> ,
	q1=>M200A1A_MixerR1_RunCmd ,
	q2=>M200A1B_MixerR1_RunCmd,
	q3=>M200A1C_MixerR1_RunCmd ,
	e1=> );

EQUIP_TYPE_3_Valve2_RA1(
	i1:=NOT reactorA1.q3 ,
	i2:= reactorA1.q3,
	s1:= XV221A_LimeValveR1_CloseStat,
	s2:= XV221A_LimeValveR1_OpenStat,
	c1=> ,
	q1=>XV221A_LimeValveR1_CloseCmd ,
	q2=>XV221A_LimeValveR1_OpenCmd );

EQUIP_TYPE_3_Valve3_RA1(
	i1:=NOT reactorA1.q4 ,
	i2:= reactorA1.q4,
	s1:= XV211A_AlumValveR1_CloseStat,
	s2:= XV211A_AlumValveR1_OpenStat,
	c1=> ,
	q1=>XV211A_AlumValveR1_CloseCmd ,
	q2=>XV211A_AlumValveR1_OpenCmd );

EQUIP_TYPE_3_Valve4_RA1(
	i1:=NOT reactorA1.q5 ,
	i2:= reactorA1.q5,
	s1:=XV201A_AirBlowerValveR1_CloseStat ,
	s2:=XV201A_AirBlowerValveR1_OpenStat ,
	c1=> ,
	q1=>XV201A_AirBlowerValveR1_CloseCmd ,
	q2=>XV201A_AirBlowerValveR1_OpenCmd );

EQUIP_TYPE_9_Valve5_RA1(
	i1:= NOT reactorA1.q7 ,
	i2:=reactorA1.q7 ,
	s1:=XV241A_SludgeValveR1_CloseStat ,
	s2:=XV241A_SludgeValveR1_OpenStat ,
	c1=> ,
	q1=>XV241A_SludgeValveR1_CloseCmd ,
	q2=>XV241A_SludgeValveR1_OpenCmd );

EQUIP_TYPE_10_Dec_RA1(
	i1:=reactorA1.q8 ,
	i2:= reactorA1.q9,
	r1:= reset_dec_RA1,
	s1:= XV261A_DecanterR1_EStopStat,
	s2:= XV261A_DecanterR1_FwdStat,
	s3:= XV261A_DecanterR1_OverloadStat,
	s4:= XV261A_DecanterR1_OverloadStat,
	s5:= XV261A_DecanterR1_RvsStat,
	q1=> XV261A_DecanterR1_RvsCmd,
	q2=>XV261A_DecanterR1_FwdCmd ,
	e1=> );




EQUIP_TYPE_3_Valva1_RA2(
	i1:=NOT reactorA2.q1 ,
	i2:=reactorA2.q1 ,
	s1:=XV206A_SBRValveR2_CloseStat ,
	s2:=XV206A_SBRValveR2_OpenStat ,
	c1=> ,
	q1=>XV206A_SBRValveR2_CloseCmd ,
	q2=>XV206A_SBRValveR2_OpenCmd);

EQUIP_TYPE_8_MIXER_A2(
	i1:= NOT reactorA2.q2,
	i2:= reactorA2.q2,
	sa1:=M200A2A_MixerR2_EStopStat,
	sa2:=M200A2A_MixerR2_IncompleteStat ,
	sa3:=M200A2A_MixerR2_LocalRemoteStat ,
	sa4:=M200A2A_MixerR2_OverloadStat ,
	sa5:=M200A2A_MixerR2_RunStat ,
	sb1:=M200A2B_MixerR2_EStopStat,
	sb2:=M200A2B_MixerR2_IncompleteStat ,
	sb3:=M200A2B_MixerR2_LocalRemoteStat ,
	sb4:=M200A2B_MixerR2_OverloadStat ,
	sb5:=M200A2B_MixerR2_RunStat ,
	sc1:=M200A2C_MixerR2_EStopStat,
	sc2:=M200A2C_MixerR2_IncompleteStat ,
	sc3:=M200A2C_MixerR2_LocalRemoteStat ,
	sc4:=M200A2C_MixerR2_OverloadStat ,
	sc5:=M200A2C_MixerR2_RunStat ,
	c1=> ,
	q1=>M200A2A_MixerR2_RunCmd ,
	q2=>M200A2B_MixerR2_RunCmd,
	q3=>M200A2C_MixerR2_RunCmd ,
	e1=> );

EQUIP_TYPE_3_Valve2_RA2(
	i1:=NOT reactorA2.q3 ,
	i2:= reactorA2.q3,
	s1:= XV222A_LimeValveR2_CloseStat,
	s2:= XV222A_LimeValveR2_OpenStat,
	c1=> ,
	q1=>XV222A_LimeValveR2_CloseCmd ,
	q2=>XV222A_LimeValveR2_OpenCmd );

EQUIP_TYPE_3_Valve3_RA2(
	i1:=NOT reactorA2.q4 ,
	i2:= reactorA2.q4,
	s1:= XV212A_AlumValveR2_CloseStat,
	s2:= XV212A_AlumValveR2_OpenStat,
	c1=> ,
	q1=>XV212A_AlumValveR2_CloseCmd ,
	q2=>XV212A_AlumValveR2_OpenCmd );

EQUIP_TYPE_3_Valve4_RA2(
	i1:=NOT reactorA2.q5 ,
	i2:= reactorA2.q5,
	s1:=XV202A_AirBlowerValveR2_CloseStat ,
	s2:=XV202A_AirBlowerValveR2_OpenStat ,
	c1=> ,
	q1=>XV202A_AirBlowerValveR2_CloseCmd ,
	q2=>XV202A_AirBlowerValveR2_OpenCmd );


EQUIP_TYPE_9_Valve5_RA2(
	i1:= NOT reactorA2.q7 ,
	i2:=reactorA2.q7 ,
	s1:=XV242A_SludgeValveR2_CloseStat ,
	s2:=XV242A_SludgeValveR2_OpenStat ,
	c1=> ,
	q1=>XV242A_SludgeValveR2_CloseCmd ,
	q2=>XV242A_SludgeValveR2_OpenCmd );

EQUIP_TYPE_10_Dec_RA2(
	i1:=reactorA2.q8 ,
	i2:= reactorA2.q9,
	r1:= reset_dec_RA2,
	s1:= XV262A_DecanterR2_EStopStat,
	s2:= XV262A_DecanterR2_FwdStat,
	s3:= XV262A_DecanterR2_OverloadStat,
	s4:= XV262A_DecanterR2_OverloadStat,
	s5:= XV262A_DecanterR2_RvsStat,
	q1=> XV262A_DecanterR2_RvsCmd,
	q2=>XV262A_DecanterR2_FwdCmd ,
	e1=> );




EQUIP_TYPE_3_Valva1_RA3(
	i1:=NOT reactorA3.q1 ,
	i2:=reactorA3.q1 ,
	s1:=XV207A_SBRValveR3_CloseStat ,
	s2:=XV207A_SBRValveR3_OpenStat ,
	c1=> ,
	q1=>XV207A_SBRValveR3_CloseCmd ,
	q2=>XV207A_SBRValveR3_OpenCmd);

EQUIP_TYPE_8_MIXER_A3(
	i1:= NOT reactorA3.q2,
	i2:= reactorA3.q2,
	sa1:=M200A3A_MixerR3_EStopStat,
	sa2:=M200A3A_MixerR3_IncompleteStat ,
	sa3:=M200A3A_MixerR3_LocalRemoteStat ,
	sa4:=M200A3A_MixerR3_OverloadStat ,
	sa5:=M200A3A_MixerR3_RunStat ,
	sb1:=M200A3B_MixerR3_EStopStat,
	sb2:=M200A3B_MixerR3_IncompleteStat ,
	sb3:=M200A3B_MixerR3_LocalRemoteStat ,
	sb4:=M200A3B_MixerR3_OverloadStat ,
	sb5:=M200A3B_MixerR3_RunStat ,
	sc1:=M200A3C_MixerR3_EStopStat,
	sc2:=M200A3C_MixerR3_IncompleteStat ,
	sc3:=M200A3C_MixerR3_LocalRemoteStat ,
	sc4:=M200A3C_MixerR3_OverloadStat ,
	sc5:=M200A3C_MixerR3_RunStat ,
	c1=> ,
	q1=>M200A3A_MixerR3_RunCmd ,
	q2=>M200A3B_MixerR3_RunCmd,
	q3=>M200A3C_MixerR3_RunCmd ,
	e1=> );

EQUIP_TYPE_3_Valve2_RA3(
	i1:=NOT reactorA3.q3 ,
	i2:= reactorA3.q3,
	s1:= XV223A_LimeValveR3_CloseStat,
	s2:= XV223A_LimeValveR3_OpenStat,
	c1=> ,
	q1=>XV223A_LimeValveR3_CloseCmd ,
	q2=>XV223A_LimeValveR3_OpenCmd );

EQUIP_TYPE_3_Valve3_RA3(
	i1:=NOT reactorA3.q4 ,
	i2:= reactorA3.q4,
	s1:= XV213A_AlumValveR3_CloseStat,
	s2:= XV213A_AlumValveR3_OpenStat,
	c1=> ,
	q1=>XV213A_AlumValveR3_CloseCmd ,
	q2=>XV213A_AlumValveR3_OpenCmd );

EQUIP_TYPE_3_Valve4_RA3(
	i1:=NOT reactorA3.q5 ,
	i2:= reactorA3.q5,
	s1:=XV203A_AirBlowerValveR3_CloseStat ,
	s2:=XV203A_AirBlowerValveR3_OpenStat ,
	c1=> ,
	q1=>XV203A_AirBlowerValveR3_CloseCmd ,
	q2=>XV203A_AirBlowerValveR3_OpenCmd );


EQUIP_TYPE_9_Valve5_RA3(
	i1:= NOT reactorA3.q7 ,
	i2:=reactorA3.q7 ,
	s1:=XV243A_SludgeValveR3_CloseStat ,
	s2:=XV243A_SludgeValveR3_OpenStat ,
	c1=> ,
	q1=>XV243A_SludgeValveR3_CloseCmd ,
	q2=>XV243A_SludgeValveR3_OpenCmd );

EQUIP_TYPE_10_Dec_RA3(
	i1:=reactorA3.q8 ,
	i2:= reactorA3.q9,
	r1:= reset_dec_RA3,
	s1:= XV263A_DecanterR3_EStopStat,
	s2:= XV263A_DecanterR3_FwdStat,
	s3:= XV263A_DecanterR3_OverloadStat,
	s4:= XV263A_DecanterR3_OverloadStat,
	s5:= XV263A_DecanterR3_RvsStat,
	q1=> XV263A_DecanterR3_RvsCmd,
	q2=>XV263A_DecanterR3_FwdCmd ,
	e1=> );



EQUIP_TYPE_3_Valva1_RA4(
	i1:=NOT reactorA4.q1 ,
	i2:=reactorA4.q1 ,
	s1:=XV208A_SBRValveR4_CloseStat ,
	s2:=XV208A_SBRValveR4_OpenStat ,
	c1=> ,
	q1=>XV208A_SBRValveR4_CloseCmd ,
	q2=>XV208A_SBRValveR4_OpenCmd);

EQUIP_TYPE_8_MIXER_A4(
	i1:= NOT reactorA4.q2,
	i2:= reactorA4.q2,
	(*sa1:=M200A4A_MixerR4_EStopStat,*)
	sa2:=M200A4A_MixerR4_IncompleteStat ,
	sa3:=M200A4A_MixerR4_LocalRemoteStat ,
	sa4:=M200A4A_MixerR4_OverloadStat ,
	sa5:=M200A4A_MixerR4_RunStat ,
	(*sb1:=M200A4B_MixerR4_EStopStat,*)
	sb2:=M200A4B_MixerR4_IncompleteStat ,
	sb3:=M200A4B_MixerR4_LocalRemoteStat ,
	sb4:=M200A4B_MixerR4_OverloadStat ,
	sb5:=M200A4B_MixerR4_RunStat ,
	(*sc1:=M200A4C_MixerR4_EStopStat,*)
	sc2:=M200A4C_MixerR4_IncompleteStat ,
	sc3:=M200A4C_MixerR4_LocalRemoteStat ,
	sc4:=M200A4C_MixerR4_OverloadStat ,
	sc5:=M200A4C_MixerR4_RunStat ,
	c1=> ,
	q1=>M200A4A_MixerR4_RunCmd ,
	q2=>M200A4B_MixerR4_RunCmd,
	q3=>M200A4C_MixerR4_RunCmd ,
	e1=> );

EQUIP_TYPE_3_Valve2_RA4(
	i1:=NOT reactorA4.q3 ,
	i2:= reactorA4.q3,
	s1:= XV224A_LimeValveR4_CloseStat,
	s2:= XV224A_LimeValveR4_OpenStat,
	c1=> ,
	q1=>XV224A_LimeValveR4_CloseCmd ,
	q2=>XV224A_LimeValveR4_OpenCmd );

EQUIP_TYPE_3_Valve3_RA4(
	i1:=NOT reactorA4.q4 ,
	i2:= reactorA4.q4,
	s1:= XV214A_AlumValveR4_CloseStat,
	s2:= XV214A_AlumValveR4_OpenStat,
	c1=> ,
	q1=>XV214A_AlumValveR4_CloseCmd ,
	q2=>XV214A_AlumValveR4_OpenCmd );

EQUIP_TYPE_3_Valve4_RA4(
	i1:=NOT reactorA4.q5 ,
	i2:= reactorA4.q5,
	s1:=XV204A_AirBlowerValveR4_CloseStat ,
	s2:=XV204A_AirBlowerValveR4_OpenStat ,
	c1=> ,
	q1=>XV204A_AirBlowerValveR4_CloseCmd ,
	q2=>XV204A_AirBlowerValveR4_OpenCmd );

EQUIP_TYPE_9_Valve5_RA4(
	i1:= NOT reactorA4.q7 ,
	i2:=reactorA4.q7 ,
	s1:=XV244A_SludgeValveR4_CloseStat ,
	s2:=XV244A_SludgeValveR4_OpenStat ,
	c1=> ,
	q1=>XV244A_SludgeValveR4_CloseCmd ,
	q2=>XV244A_SludgeValveR4_OpenCmd );

EQUIP_TYPE_10_Dec_RA4(
	i1:=reactorA4.q8 ,
	i2:= reactorA4.q9,
	r1:= reset_dec_RA4,
	s1:= XV264A_DecanterR4_EStopStat,
	s2:= XV264A_DecanterR4_FwdStat,
	s3:= XV264A_DecanterR4_OverloadStat,
	s4:= XV264A_DecanterR4_OverloadStat,
	s5:= XV264A_DecanterR4_RvsStat,
	q1=> XV264A_DecanterR4_RvsCmd,
	q2=>XV264A_DecanterR4_FwdCmd ,
	e1=> );
END_ACTION
ACTION reactorB:
(*REACTOR A*)

reactorB1(
	op:= OPR1B_ReactorStatus,
	res_fill:=Fill_selectorB.q1 ,
	i1:= LSH201B1_LevelSensorR1 ,
	alum_time:= Alum_reactorB1,
	res_aeration:= Aerate_selectorB.q1,
	ph1:=PHT201B1_pHlevelR1 ,
	res_decanting:=Decant_selectorB.q1 ,
	r1:=resumeAlumB1 ,
	i2:=LSHH501B_SludgeStorage ,
	i3:=HR201B1_DecantHighLevelR1 ,
	i4:=LR201B1_DecantLowLevelR1 ,
	req_fill=> ,
	q1=> ,
	q2=> ,
	q4=> ,
	q3=> ,
	q5=> ,
	q6=> ,
	req_aeration=> ,
	e1=> ,
	q7=> ,
	q8=> ,
	m1=> ,
	req_settle=> ,
	req_decanting=> ,
	q9=> );

reactorB2(
	op:= OPR2B_ReactorStatus,
	res_fill:=Fill_selectorB.q2 ,
	i1:= LSH201B2_LevelSensorR2 ,
	alum_time:= Alum_reactorB2,
	res_aeration:= Aerate_selectorB.q2,
	ph1:=PHT201B2_pHlevelR2 ,
	res_decanting:=Decant_selectorB.q2 ,
	r1:=resumeAlumB2 ,
	i2:=LSHH501B_SludgeStorage ,
	i3:=HR201B2_DecantHighLevelR2 ,
	i4:=LR201B2_DecantLowLevelR2 ,
	req_fill=> ,
	q1=> ,
	q2=> ,
	q4=> ,
	q3=> ,
	q5=> ,
	q6=> ,
	req_aeration=> ,
	e1=> ,
	q7=> ,
	q8=> ,
	m1=> ,
	req_settle=> ,
	req_decanting=> ,
	q9=> );

reactorB3(
	op:= OPR3B_ReactorStatus,
	res_fill:=Fill_selectorB.q3 ,
	i1:= LSH201B3_LevelSensorR3 ,
	alum_time:= Alum_reactorB3,
	res_aeration:= Aerate_selectorB.q3,
	ph1:=PHT201B3_pHlevelR3 ,
	res_decanting:=Decant_selectorB.q3 ,
	r1:=resumeAlumB3 ,
	i2:=LSHH501B_SludgeStorage ,
	i3:=HR201B3_DecantHighLevelR3 ,
	i4:=LR201B3_DecantLowLevelR3 ,
	req_fill=> ,
	q1=> ,
	q2=> ,
	q4=> ,
	q3=> ,
	q5=> ,
	q6=> ,
	req_aeration=> ,
	e1=> ,
	q7=> ,
	q8=> ,
	m1=> ,
	req_settle=> ,
	req_decanting=> ,
	q9=> );

reactorB4(
	op:= OPR4B_ReactorStatus,
	res_fill:=Fill_selectorB.q4 ,
	i1:= LSH201B4_LevelSensorR4 ,
	alum_time:= Alum_reactorB4,
	res_aeration:= Aerate_selectorB.q4,
	ph1:=PHT201B4_pHlevelR4 ,
	res_decanting:=Decant_selectorB.q4 ,
	r1:=resumeAlumB4 ,
	i2:=LSHH501B_SludgeStorage ,
	i3:=HR201B4_DecantHighLevelR4 ,
	i4:=LR201B4_DecantLowLevelR4 ,
	req_fill=> ,
	q1=> ,
	q2=> ,
	q4=> ,
	q3=> ,
	q5=> ,
	q6=> ,
	req_aeration=> ,
	e1=> ,
	q7=> ,
	q8=> ,
	m1=> ,
	req_settle=> ,
	req_decanting=> ,
	q9=> );

fill_selectorB(
	i1:=ReactorB1.req_fill ,
	i2:=ReactorB2.req_fill ,
	i3:=ReactorB3.req_fill ,
	i4:=ReactorB4.req_fill,
	q1=> ,
	q2=> ,
	q3=> ,
	q4=> ,
	c1=> );

aerate_selectorB(
	i1:=ReactorB1.req_aeration,
	i2:=ReactorB2.req_aeration ,
	i3:=ReactorB3.req_aeration ,
	i4:=ReactorB4.req_aeration ,
	available:=2 ,
	q1=> ,
	q2=> ,
	q3=> ,
	q4=>);

sbr_airblower_B(
	sa1:= B201B1_AirBlowerS2_EStopStat,
	sa2:= B201B1_AirBlowerS2_IncompleteStat,
	sa3:= B201B1_AirBlowerS2_LocalRemoteStat,
	sa4:= B201B1_AirBlowerS2_OverloadStat,
	sa5:= B201B1_AirBlowerS2_RunStat,
	sb1:= B201B2_AirBlowerS2_EStopStat,
	sb2:= B201B2_AirBlowerS2_IncompleteStat,
	sb3:= B201B2_AirBlowerS2_LocalRemoteStat,
	sb4:= B201B2_AirBlowerS2_OverloadStat,
	sb5:= B201B2_AirBlowerS2_RunStat,
	sc1:= B201B3_AirBlowerS2_EStopStat,
	sc2:= B201B3_AirBlowerS2_IncompleteStat,
	sc3:= B201B3_AirBlowerS2_LocalRemoteStat,
	sc4:= B201B3_AirBlowerS2_OverloadStat,
	sc5:= B201B3_AirBlowerS2_RunStat,
	req:= aerate_selectorA.taken,
	q1=> B201B1_AirBlowerS2_RunCmd,
	q2=> B201B2_AirBlowerS2_RunCmd,
	q3=> B201B3_AirBlowerS2_RunCmd);

decant_selectorB(
	i1:=  ReactorB1.req_decanting,
	i2:=  ReactorB2.req_decanting,
	i3:=  ReactorB3.req_decanting,
	i4:=  ReactorB4.req_decanting,
	q1=> ,
	q2=> ,
	q3=> ,
	q4=> ,
	c1=> );


